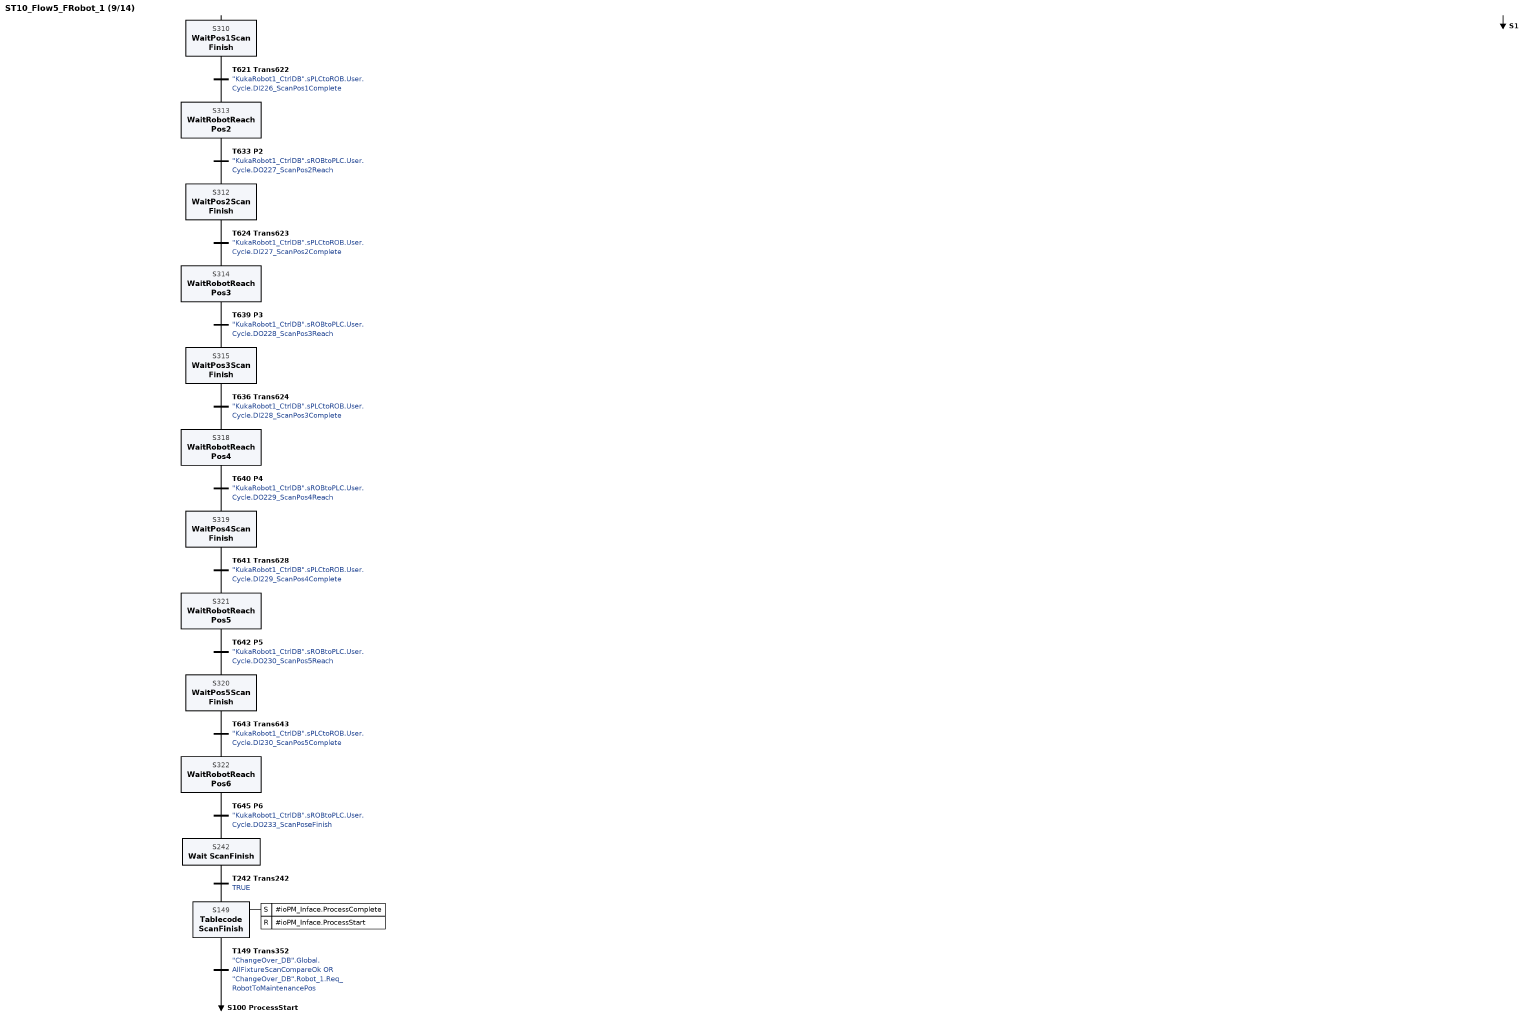
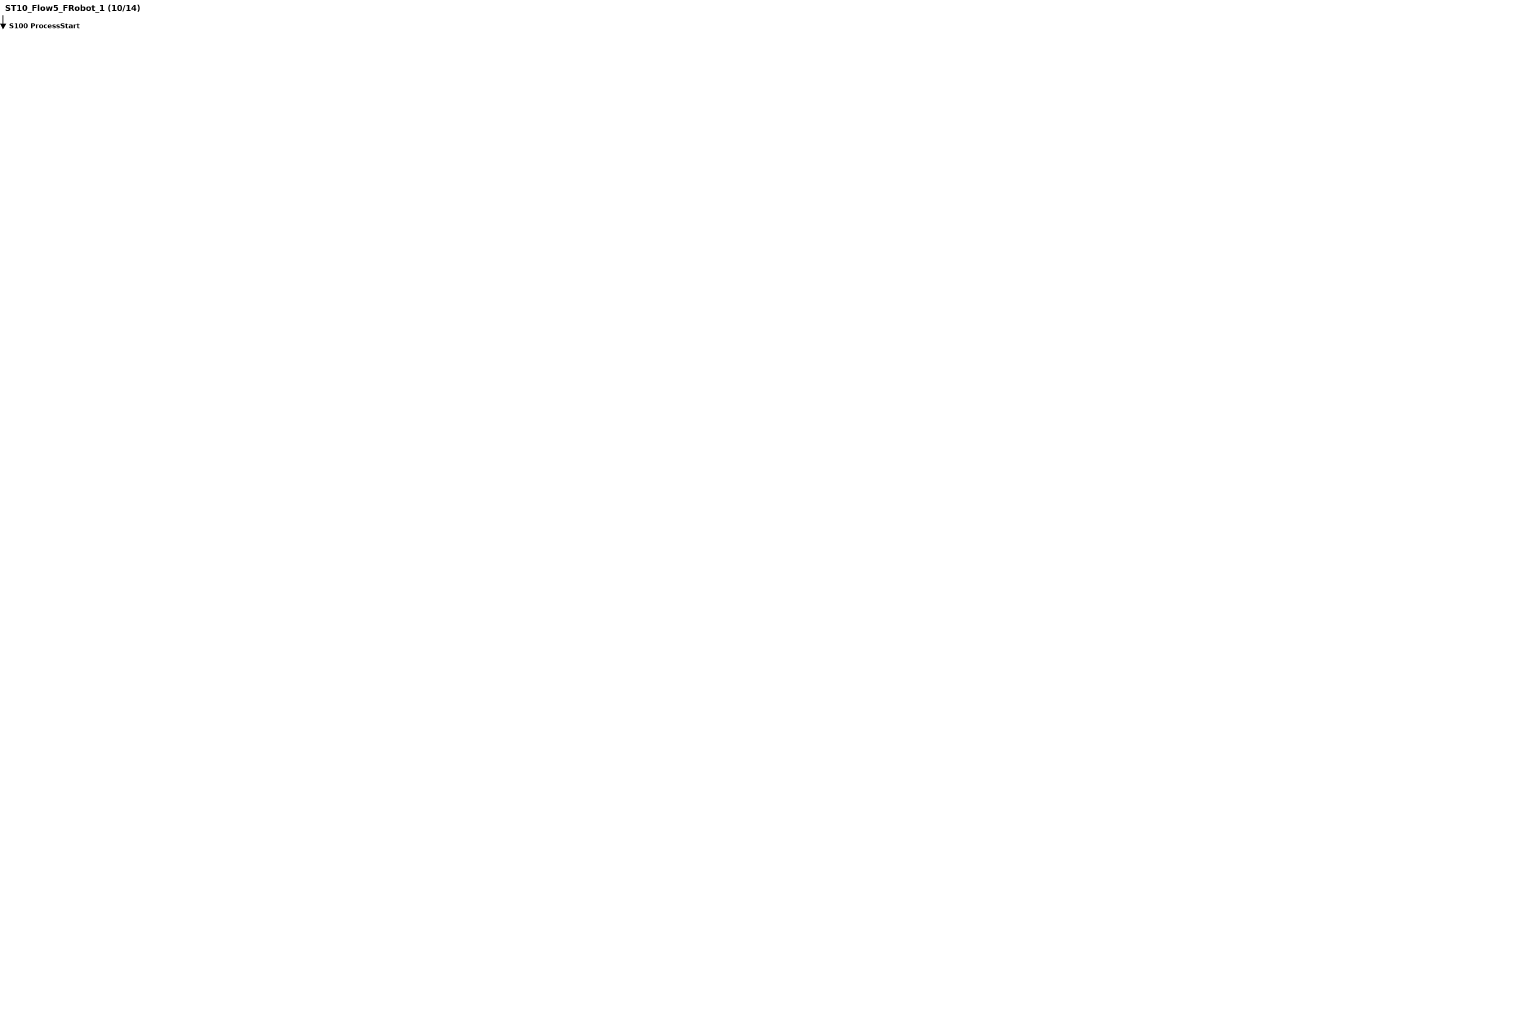
   // permanent pre-instructions
   NETWORK 1
      #TON[10].TON(IN := "AlwaysTRUE" AND "Station_Sys".Alarm.ImmediatelyStop, PT := T#300ms);
      #ioPM_Inface.AlarmImdilyStop := #TON[10].Q;
      #ioPM_Inface.AlarmCycleStop := "AlwaysTRUE" AND "Station_Sys".Alarm.CycleStop;
   NETWORK 2
      IF NOT False THEN
          #sCtrlMode(iSysInface := #iSysInface, ioPM_Inface := #ioPM_Inface, ioGraphCtrl := #RT_DATA.MOP);   // "SysFlowCtrlGraph"
      END_IF;
   NETWORK 3
      #TON[0].TON(IN := "AlwaysTRUE" AND "iA-Rotating product Check", PT := t#500ms);   // 工位11有托盘
      #TON[1].TOF(IN := "AlwaysTRUE" AND NOT "iA-Rotating product Check", PT := T#300ms);   // 工位无托盘
      #TON[2].TON(IN := "AlwaysTRUE", PT := T#300ms);
      #TON[3].TON(IN := "AlwaysTRUE", PT := T#300ms);
      #TON[4].TON(IN := "AlwaysTRUE", PT := T#300ms);
      #TON[5].TON(IN := "AlwaysTRUE", PT := T#300ms);
   NETWORK 4
      #前站站号 := 345;
      #本站站号 := 350;

   // sequencer 1: S01-S99 初始化
   INITIAL_STEP F5_Initial:   // S1, max time T#10S, warning time T#7S
              S    #ioPM_Inface.InitialRun
              R    #ioPM_Inface.InitialOK
              R    #ioPM_Inface.WaitRunning
              R    #ioPM_Inface.Running
              R    #ioPM_Inface.UnPause
              R    "Station_Sys".Cmd.Calibration
              R    "Station_Sys".Cmd.ChangeOver
                   //"ST350_Sys".Cmd.DryRun
              R    "Station_Sys".Cmd.Reserve
              R    "Station_Sys".Cmd.OneCycle
              R    "AutoProcessControl".Robot_1.GluePutFlag
              R    "AutoProcessControl".Robot_1.NGPutFlag
              R    #ioPM_Inface.ProcessComplete
              R    #ioPM_Inface.ProcessStart
          S1  R    "ChangeOver_DB".Robot_1.MaintenancePosReqSelFlag
                   //"Robot_DB".Robot_1.MasteringTest_Req
                   //"Robot_DB".Robot_1.BrakeTest_Req
   END_STEP
   TRANSITION Trans1 FROM F5_Initial TO S2   // T1
      := #iSysInface.Ready;
   END_TRANSITION
   STEP S2:   // S2, max time T#10S, warning time T#7S
   END_STEP
   TRANSITION Trans2 FROM S2 TO S3   // T2
      := TRUE;
   END_TRANSITION
   STEP RobotSpeed:   // S4, max time T#10S, warning time T#7S
              N    "KukaRobot1_CtrlDB".iSpeedValue:=20
   END_STEP
   TRANSITION Trans3 FROM RobotSpeed TO S5_MESInitial   // T3
      := "KukaRobot1_CtrlDB".iSpeedValue = 20;
   END_TRANSITION
   STEP S5_MESInitial:   // S5, max time T#10S, warning time T#7S
   END_STEP
   TRANSITION Trans325 FROM S5_MESInitial TO "RobotManuallyMoved?"   // T4
      := TRUE;
   END_TRANSITION
   STEP S10_InitialFinish:   // S10, max time T#10S, warning time T#7S
              S    #ioPM_Inface.InitialOK
   END_STEP
   TRANSITION Trans102 FROM S10_InitialFinish TO ProcessStart   // T10, jump
      := #ioPM_Inface.Running;
   END_TRANSITION
   STEP S3:   // S3, max time T#10S, warning time T#7S
   END_STEP
   TRANSITION Trans613 FROM S3 TO RobotSpeed   // T607
      := TRUE;
   END_TRANSITION
   STEP S8:   // S8, max time T#10S, warning time T#7S
   END_STEP
   TRANSITION Trans10 FROM S8 TO S9   // T8
      := TRUE;
   END_TRANSITION
   STEP S9:   // S9, max time T#10S, warning time T#7S
   END_STEP
   TRANSITION Trans7 FROM S9 TO S10_InitialFinish   // T9
      := TRUE;
   END_TRANSITION
   STEP "RobotReady?":   // S311, max time T#10S, warning time T#7S
   END_STEP
   TRANSITION Trans606 FROM "RobotReady?" TO RobotStart   // T606
      := "KukaRobot1_CtrlDB".sROBtoPLC.Sys.SO.ALARM_STOP AND "KukaRobot1_CtrlDB".sROBtoPLC.Sys.SO.EXT AND NOT "KukaRobot1_CtrlDB".oStartComplete;
   END_TRANSITION
   STEP RobotStart:   // S316, max time T#10S, warning time T#7S
              N    "KukaRobot1_CtrlDB".ioAutoStart
   END_STEP
   TRANSITION Trans608 FROM RobotStart TO WaitRobotStartHome   // T608
      := "KukaRobot1_CtrlDB".oReady AND "KukaRobot1_CtrlDB".oStartComplete;
   END_TRANSITION
   STEP RobotHome:   // S317, max time T#10S, warning time T#7S
              N    "KukaRobot1_CtrlDB".ioSrartHome
   END_STEP
   TRANSITION Trans609 FROM RobotHome TO RobotAutoCycle   // T609
      := "KukaRobot1_CtrlDB".sROBtoPLC.Sys.SO.IN_HOME AND "KukaRobot1_CtrlDB".sHMI.HomeSeqOK AND "KukaRobot1_CtrlDB".sHMI.WaitForAutoCycleStart AND NOT "KukaRobot1_CtrlDB".sHMI.GoHomeFail;
   END_TRANSITION
   STEP RobotAutoCycle:   // S329, max time T#10S, warning time T#7S
              N    "KukaRobot1_CtrlDB".ioStartAutoCycle
   END_STEP
   TRANSITION Trans612 FROM RobotAutoCycle TO GripStatusCheck   // T610
      := NOT "KukaRobot1_CtrlDB".sHMI.HomeSeqOK AND NOT "KukaRobot1_CtrlDB".sHMI.WaitForAutoCycleStart;
   END_TRANSITION
   STEP GripStatusCheck:   // S330, max time T#10S, warning time T#7S
   END_STEP
   TRANSITION Trans614 FROM GripStatusCheck TO S8   // T611
      := (("AutoProcessData".F_Robot1Grip1.PartStatus = 0) AND ("AutoProcessData".F_Robot1Grip2.PartStatus = 0) AND "iF-ROOBT1Gripper1CylinderInHP" AND NOT "iF-ROOBT1Gripper2Detection") OR (("AutoProcessData".F_Robot1Grip1.PartStatus <> 0) AND NOT "iF-ROOBT1Gripper1CylinderInHP" AND NOT "iF-ROOBT1Gripper1CylinderInWP") OR (("AutoProcessData".F_Robot1Grip2.PartStatus <> 0) AND "iF-ROOBT1Gripper2Detection");
   END_TRANSITION
   TRANSITION Trans616 FROM GripStatusCheck TO Gripe1StatusAlarm   // T613
      := (("AutoProcessData".F_Robot1Grip1.PartStatus = 0) AND NOT "iF-ROOBT1Gripper1CylinderInHP" AND NOT "iF-ROOBT1Gripper1CylinderInWP" AND NOT "ST10Cylinder".Cy[13].In.HomePositionSensor) OR (("AutoProcessData".F_Robot1Grip1.PartStatus <> 0) AND ("iF-ROOBT1Gripper1CylinderInWP" OR "ST10Cylinder".Cy[13].In.HomePositionSensor));
   END_TRANSITION
   TRANSITION Trans617 FROM GripStatusCheck TO Gripe2StatusAlarm   // T612
      := (("AutoProcessData".F_Robot1Grip2.PartStatus = 0) AND "iF-ROOBT1Gripper2Detection" AND NOT "ST10Cylinder".Cy[14].In.HomePositionSensor) OR (("AutoProcessData".F_Robot1Grip2.PartStatus <> 0) AND (NOT "iF-ROOBT1Gripper2Detection" OR "ST10Cylinder".Cy[14].In.HomePositionSensor));
   END_TRANSITION
   STEP Gripe1StatusAlarm:   // S331, max time T#10S, warning time T#7S
          S1  S    "ST10_DeviceError".F.Robot_1.Grip1Error
   END_STEP
   TRANSITION Trans615 FROM Gripe1StatusAlarm TO GripStatusCheck   // T614, jump
      := #iSysInface.Reset;
   END_TRANSITION
   STEP Gripe2StatusAlarm:   // S332, max time T#10S, warning time T#7S
          S1  S    "ST10_DeviceError".F.Robot_1.Grip2Error
   END_STEP
   TRANSITION Trans620 FROM Gripe2StatusAlarm TO GripStatusCheck   // T615, jump
      := #iSysInface.Reset;
   END_TRANSITION
   STEP WaitRobotStartHome:   // S381, max time T#10S, warning time T#7S
   END_STEP
   TRANSITION Trans695 FROM WaitRobotStartHome TO RobotHome   // T695
      := "KukaRobot1_CtrlDB".sROBtoPLC.User.Home.DO161_WaitForHomeSeqStart;
   END_TRANSITION
   STEP "RobotManuallyMoved?":   // S382, max time T#10S, warning time T#7S
   END_STEP
   TRANSITION Trans696 FROM "RobotManuallyMoved?" TO "RobotReady?"   // T696
      := NOT "KukaRobot1_CtrlDB".sPLCtoROB.User.Home.DI169_RobotMoved AND NOT "ST10_DeviceError".F.Robot_1.ManualMoved;
   END_TRANSITION

   // sequencer 2: S100-S199 等待到位
   STEP ProcessStart:   // S100, max time T#10S, warning time T#7S
      // 自动等待开始运行
              R    #ioPM_Inface.InitialRun
              R    #ioPM_Inface.ProcessComplete
              R    #ioPM_Inface.ProcessStart
              S    #ioPM_Inface.InitialOK
              S    #ioPM_Inface.WaitRunning
          S1  N    #ioPM_Inface.ProcessResult:=0
              R    "ST10_GeneralData".FlowControl_Handshake[5].Start
              R    "ST10_GeneralData".FlowControl_Handshake[5].Done
   END_STEP
   TRANSITION Trans200 FROM ProcessStart TO FlagReset   // T100
      := NOT #ioPM_Inface.AlarmCycleStop AND #ioPM_Inface.Running AND NOT #iSysInface.Auto.RunningOver AND (NOT #iSysInface.Auto.OneCycleMode OR (#iSysInface.Auto.OneCycleMode AND #ioPM_Inface.TriggerOneCycle));
   END_TRANSITION
   STEP ScanFixtureCode:   // S110, max time T#10S, warning time T#7S
              R    #ioPM_Inface.ProcessComplete
              S    #ioPM_Inface.ProcessStart
   END_STEP
   TRANSITION Trans625 FROM ScanFixtureCode TO "Tablecode Scan"   // T110, jump
      := TRUE;
   END_TRANSITION
   STEP RobotTaskSelect:   // S333, max time T#10S, warning time T#7S
   END_STEP
   TRANSITION Trans621 FROM RobotTaskSelect TO ScanFixtureCode   // T333
      := NOT "AutoProcessData".GlobalData.Robot1GripperCodeOKFlag AND ("AutoProcessData".F_Robot1Grip1.PartStatus = 0) AND "ST10Cylinder".Cy[13].In.HomePositionSensor AND "AutoProcessControl".Robot_1.GripScanRequest AND NOT "PalletNGData".LoadingNGPallet.OpenFlag AND NOT "ChangeOver_DB".Robot_1.MaintenancePosReqSelFlag AND NOT "Robot_DB".Robot_1.MasteringTest_Req AND NOT "Robot_DB".Robot_1.BrakeTest_Req;
   END_TRANSITION
   TRANSITION Trans630 FROM RobotTaskSelect TO PutBuffer   // T620
      := ("AutoProcessData".F_Robot1Grip1.PartStatus = 100) AND NOT "iF-ROOBT1Gripper1CylinderInHP" AND NOT "iF-ROOBT1Gripper1CylinderInWP" AND NOT "ST10Cylinder".Cy[13].In.HomePositionSensor AND "AutoProcessControl".A_ScanRotary.Robot1PutPrimit AND NOT "PalletNGData".LoadingNGPallet.OpenFlag AND NOT "ChangeOver_DB".Robot_1.MaintenancePosReqSelFlag;
   END_TRANSITION
   TRANSITION Trans632 FROM RobotTaskSelect TO PickTable   // T625
      := (NOT "AutoProcessControl".Robot_1.ClearPart OR (("AutoProcessControl".B_Press_1.Robot1PutRingPrimit OR ("AutoProcessData".A_ScanRotate.PartStatus = 199)) AND "AutoProcessControl".Robot_1.ClearPart)) AND ("AutoProcessData".F_Robot1Grip1.PartStatus = 0) AND "iF-ROOBT1Gripper1CylinderInHP" AND ("AutoProcessData".F_Robot1Grip2.PartStatus = 0) AND NOT "iF-ROOBT1Gripper2Detection" AND "AutoProcessControl".A_Table_1Loading.Robot1PickPrimit AND NOT "PalletNGData".LoadingNGPallet.OpenFlag AND NOT "ChangeOver_DB".Robot_1.MaintenancePosReqSelFlag AND NOT "Robot_DB".Robot_1.MasteringTest_Req AND NOT "Robot_DB".Robot_1.BrakeTest_Req;
   END_TRANSITION
   TRANSITION Trans633 FROM RobotTaskSelect TO ScanRing   // T627
      := ("AutoProcessData".F_Robot1Grip2.PartStatus = 100) AND ("iF-ROOBT1Gripper2Detection" OR "AlwaysTRUE") AND NOT "ST10Cylinder".Cy[14].In.HomePositionSensor AND NOT "KukaRobot1_CtrlDB".sPLCtoROB.User.Cycle.DI261_RingScanReq AND NOT "ChangeOver_DB".Global.ManualModeFlag AND NOT "ChangeOver_DB".Global.ChangeOverSelected AND NOT "PalletNGData".LoadingNGPallet.OpenFlag AND NOT "ChangeOver_DB".Robot_1.MaintenancePosReqSelFlag AND NOT "Robot_DB".Robot_1.MasteringTest_Req AND NOT "Robot_DB".Robot_1.BrakeTest_Req;
   END_TRANSITION
   TRANSITION Trans635 FROM RobotTaskSelect TO PickBuffer   // T629
      := ((("AutoProcessData".F_Robot1Grip2.PartStatus = 199) AND ("iF-ROOBT1Gripper2Detection" OR "AlwaysTRUE")) OR (("AutoProcessData".F_Robot1Grip2.PartStatus = 0) AND ("AutoProcessData".A_ScanRotate.PartStatus = 151))) AND ("AutoProcessData".F_Robot1Grip1.PartStatus = 0) AND "iF-ROOBT1Gripper1CylinderInHP" AND ("AutoProcessData".B_Press1.PartStatus = 0) AND NOT "PalletNGData".LoadingNGPallet.OpenFlag AND "AutoProcessControl".A_ScanRotary.Robot1PickPrimit AND NOT "ChangeOver_DB".Robot_1.MaintenancePosReqSelFlag AND NOT "Robot_DB".Robot_1.MasteringTest_Req AND NOT "Robot_DB".Robot_1.BrakeTest_Req;
   END_TRANSITION
   TRANSITION Trans675 FROM RobotTaskSelect TO "NG1Put_1/Press"   // T674
      := ("AutoProcessData".F_Robot1Grip1.PartStatus >= 250) AND ("AutoProcessData".F_Robot1Grip1.PartStatus <= 260) AND NOT "iF-ROOBT1Gripper1CylinderInHP" AND NOT "iF-ROOBT1Gripper1CylinderInWP" AND NOT "ST10Cylinder".Cy[13].In.HomePositionSensor AND "AutoProcessControl".NG_1.Robot1PutPrimit_1 AND NOT "PalletNGData".LoadingNGPallet.OpenFlag AND NOT "ChangeOver_DB".Robot_1.MaintenancePosReqSelFlag;
   END_TRANSITION
   TRANSITION Trans750 FROM RobotTaskSelect TO "NG1Put_2/ShaftScan"   // T757
      := ("AutoProcessData".F_Robot1Grip1.PartStatus >= 150) AND ("AutoProcessData".F_Robot1Grip1.PartStatus <= 160) AND NOT "iF-ROOBT1Gripper1CylinderInHP" AND NOT "iF-ROOBT1Gripper1CylinderInWP" AND "AutoProcessControl".NG_1.Robot1PutPrimit_2 AND NOT "PalletNGData".LoadingNGPallet.OpenFlag AND NOT "ChangeOver_DB".Robot_1.MaintenancePosReqSelFlag;
   END_TRANSITION
   TRANSITION Trans751 FROM RobotTaskSelect TO "NG1Put_3/RingScan"   // T751
      := ((("AutoProcessData".F_Robot1Grip2.PartStatus >= 150) AND ("AutoProcessData".F_Robot1Grip2.PartStatus <= 160)) OR ("ChangeOver_DB".Global.ManualModeFlag AND ("AutoProcessData".F_Robot1Grip2.PartStatus = 100))) AND ("iF-ROOBT1Gripper2Detection" OR "AlwaysTRUE") AND NOT "ST10Cylinder".Cy[14].In.HomePositionSensor AND "AutoProcessControl".NG_1.Robot1PutPrimit_3 AND NOT "PalletNGData".LoadingNGPallet.OpenFlag AND NOT "ChangeOver_DB".Robot_1.MaintenancePosReqSelFlag;
   END_TRANSITION
   TRANSITION Trans691 FROM RobotTaskSelect TO Grip1SensorError   // T691
      := ((("AutoProcessData".F_Robot1Grip1.PartStatus <> 0) AND "iF-ROOBT1Gripper1CylinderInWP") OR (("AutoProcessData".F_Robot1Grip1.PartStatus = 0) AND NOT "iF-ROOBT1Gripper1CylinderInHP")) AND (#RobotTaskSelect.T > t#3000MS) AND NOT "ChangeOver_DB".Robot_1.MaintenancePosReqSelFlag;
   END_TRANSITION
   TRANSITION Trans692 FROM RobotTaskSelect TO Grip2SensorError   // T692
      := ((("AutoProcessData".F_Robot1Grip2.PartStatus <> 0) AND NOT "iF-ROOBT1Gripper2Detection") OR (("AutoProcessData".F_Robot1Grip2.PartStatus = 0) AND "iF-ROOBT1Gripper2Detection")) AND (#RobotTaskSelect.T > t#3000MS) AND NOT "ChangeOver_DB".Robot_1.MaintenancePosReqSelFlag AND "TON".TON[74].Q;
   END_TRANSITION
   TRANSITION Trans626 FROM RobotTaskSelect TO PickPallet   // T618
      := (NOT "AutoProcessControl".Robot_1.ClearPart OR ("AutoProcessControl".Robot_1.ClearPart AND ("AutoProcessData".F_Robot1Grip2.PartStatus = 199) AND ("AutoProcessData".B_Press1.PartStatus = 0) AND "AutoProcessControl".A_ScanRotary.Robot1PutPrimit) OR "KukaRobot1_CtrlDB".sROBtoPLC.User.Cycle.DO242_SPalletPickFinish) AND NOT "ChangeOver_DB".Global.ChangeOverRequest AND NOT "ChangeOver_DB".Global.ScanFixtureFlag AND "ChangeOver_DB".Global.AllFixtureScanCompareOk AND "AutoProcessData".GlobalData.Robot2GripperCodeOKFlag AND (("AutoProcessData".F_Robot1Grip1.PartStatus = 0) OR ("AutoProcessData".F_Robot1Grip1.PartStatus = 100)) AND "iF-ROOBT1Gripper1CylinderInHP" AND "AutoProcessControl".H_ShafeLine.Robot1PickPrimit AND "AutoProcessControl".A_ScanRotary.Robot1PutPrimit AND NOT "AutoProcessControl".Global.H.EmptyPallet AND ("AutoProcessData".B_Press1.PartStatus <> 199) AND NOT "ChangeOver_DB".Global.ManualModeFlag AND NOT "ChangeOver_DB".Global.ChangeOverSelected AND NOT "PalletNGData".LoadingNGPallet.OpenFlag AND NOT "ChangeOver_DB".Robot_1.MaintenancePosReqSelFlag AND NOT "KukaRobot1_CtrlDB".sROBtoPLC.User.Safety.DO452 AND NOT "KukaRobot1_CtrlDB".sROBtoPLC.User.Safety.DO460 AND (#RobotTaskSelect.T > t#100MS);
   END_TRANSITION
   TRANSITION Trans642 FROM RobotTaskSelect TO PressPick   // T637
      := ("AutoProcessData".F_Robot1Grip1.PartStatus = 0) AND "iF-ROOBT1Gripper1CylinderInHP" AND "AutoProcessControl".B_Press_1.Robot1PickPrimit AND NOT "PalletNGData".LoadingNGPallet.OpenFlag AND NOT "ChangeOver_DB".Robot_1.MaintenancePosReqSelFlag AND NOT "Robot_DB".Robot_1.MasteringTest_Req AND NOT "Robot_DB".Robot_1.BrakeTest_Req;
   END_TRANSITION
   TRANSITION Trans672 FROM RobotTaskSelect TO GluePut   // T672
      := ("AutoProcessData".F_Robot1Grip1.PartStatus = 299) AND NOT "iF-ROOBT1Gripper1CylinderInHP" AND NOT "iF-ROOBT1Gripper1CylinderInWP" AND NOT "ST10Cylinder".Cy[13].In.HomePositionSensor AND "KukaRobot2_CtrlDB".sROBtoPLC.User.Home.DO182_Robot1Area AND NOT "KukaRobot2_CtrlDB".sROBtoPLC.User.Cycle.DO241_PickPalletInside AND NOT "KukaRobot2_CtrlDB".sROBtoPLC.User.Cycle.DO261_ScanPartInside AND NOT "KukaRobot2_CtrlDB".sROBtoPLC.User.Cycle.DO265_GluePutInside AND NOT "KukaRobot2_CtrlDB".sROBtoPLC.User.Cycle.DO269_GluePickInside AND NOT "AutoProcessControl".Robot_2.PalletPickFlag AND NOT "AutoProcessControl".Robot_2.MagnetScanFlag AND NOT "AutoProcessControl".Robot_2.GluePutFlag AND NOT "AutoProcessControl".Robot_2.GluePickFlag AND "AutoProcessControl".C_Glue.Robot1PutPrimit AND NOT "PalletNGData".LoadingNGPallet.OpenFlag AND NOT "ChangeOver_DB".Robot_1.MaintenancePosReqSelFlag AND NOT "Robot_DB".Robot_1.MasteringTest_Req AND NOT "Robot_DB".Robot_1.BrakeTest_Req;
   END_TRANSITION
   TRANSITION Trans637 FROM RobotTaskSelect TO PressShaftPut   // T631
      := ("AutoProcessData".F_Robot1Grip1.PartStatus = 199) AND NOT "iF-ROOBT1Gripper1CylinderInHP" AND NOT "iF-ROOBT1Gripper1CylinderInWP" AND NOT "ST10Cylinder".Cy[13].In.HomePositionSensor AND ("AutoProcessData".F_Robot1Grip2.PartStatus = 199) AND ("iF-ROOBT1Gripper2Detection" OR "AlwaysTRUE") AND NOT "ST10Cylinder".Cy[14].In.HomePositionSensor AND "AutoProcessControl".B_Press_1.Robot1PutShaftPrimit AND NOT "PalletNGData".LoadingNGPallet.OpenFlag AND NOT "ChangeOver_DB".Robot_1.MaintenancePosReqSelFlag AND NOT "Robot_DB".Robot_1.MasteringTest_Req AND NOT "Robot_DB".Robot_1.BrakeTest_Req;
   END_TRANSITION
   TRANSITION Trans640 FROM RobotTaskSelect TO PressRingPut   // T634
      := ("AutoProcessData".F_Robot1Grip2.PartStatus = 199) AND ("iF-ROOBT1Gripper2Detection" OR "AlwaysTRUE") AND NOT "ST10Cylinder".Cy[14].In.HomePositionSensor AND ("AutoProcessData".F_Robot1Grip1.PartStatus = 0) AND "iF-ROOBT1Gripper1CylinderInHP" AND "ST10Cylinder".Cy[13].In.HomePositionSensor AND "AutoProcessControl".B_Press_1.Robot1PutRingPrimit AND NOT "PalletNGData".LoadingNGPallet.OpenFlag AND NOT "ChangeOver_DB".Robot_1.MaintenancePosReqSelFlag AND NOT "Robot_DB".Robot_1.MasteringTest_Req AND NOT "Robot_DB".Robot_1.BrakeTest_Req;
   END_TRANSITION
   TRANSITION Trans711 FROM RobotTaskSelect TO Maintenance   // T638
      := (("iF-ROOBT1Gripper1CylinderInHP" AND NOT "iF-ROOBT1Gripper2Detection" AND ("AutoProcessData".F_Robot1Grip2.PartStatus = 0) AND ("AutoProcessData".F_Robot1Grip1.PartStatus = 0) AND "ChangeOver_DB".Robot_1.Req_RobotToMaintenancePos AND NOT "PalletNGData".LoadingNGPallet.OpenFlag) OR (NOT "AutoProcessControl".Robot_1.MaintenanceRequest AND "ChangeOver_DB".Robot_1.HMI_MaintenancePosActive)) AND NOT "Robot_DB".Robot_1.MasteringTest_Req AND NOT "Robot_DB".Robot_1.BrakeTest_Req;
   END_TRANSITION
   TRANSITION Trans900 FROM RobotTaskSelect TO Masref_test   // T900
      := ("AutoProcessData".F_Robot1Grip1.PartStatus = 0) AND "iF-ROOBT1Gripper1CylinderInHP" AND "Robot_DB".Robot_1.MasteringTest_Req;
   END_TRANSITION
   TRANSITION Trans901 FROM RobotTaskSelect TO Brake_Test   // T901
      := ("AutoProcessData".F_Robot1Grip1.PartStatus = 0) AND "iF-ROOBT1Gripper1CylinderInHP" AND "Robot_DB".Robot_1.BrakeTest_Req;
   END_TRANSITION
   STEP PressPick:   // S150, max time T#10S, warning time T#7S
              R    #ioPM_Inface.ProcessComplete
              S    #ioPM_Inface.ProcessStart
   END_STEP
   TRANSITION Trans641 FROM PressPick TO PressPickProcess   // T150, jump
      := TRUE;
   END_TRANSITION
   STEP PutBuffer:   // S120, max time T#10S, warning time T#7S
              R    #ioPM_Inface.ProcessComplete
              S    #ioPM_Inface.ProcessStart
   END_STEP
   TRANSITION Trans629 FROM PutBuffer TO PutBufferProcess   // T120, jump
      := TRUE;
   END_TRANSITION
   STEP PickTable:   // S130, max time T#10S, warning time T#7S
              R    #ioPM_Inface.ProcessComplete
              S    #ioPM_Inface.ProcessStart
   END_STEP
   TRANSITION Trans631 FROM PickTable TO PickTableProcess   // T130, jump
      := TRUE;
   END_TRANSITION
   STEP ScanRing:   // S135, max time T#10S, warning time T#7S
              R    #ioPM_Inface.ProcessComplete
              S    #ioPM_Inface.ProcessStart
   END_STEP
   TRANSITION Trans634 FROM ScanRing TO ScanRingProcess   // T135, jump
      := TRUE;
   END_TRANSITION
   STEP PickBuffer:   // S125, max time T#10S, warning time T#7S
              R    #ioPM_Inface.ProcessComplete
              S    #ioPM_Inface.ProcessStart
   END_STEP
   TRANSITION Trans636 FROM PickBuffer TO PickBufferProcess   // T125, jump
      := TRUE;
   END_TRANSITION
   STEP "NG1Put_1/Press":   // S160, max time T#10S, warning time T#7S
              S    "AutoProcessControl".Robot_1.NGPutFlag
              R    #ioPM_Inface.ProcessComplete
              S    #ioPM_Inface.ProcessStart
   END_STEP
   TRANSITION Trans676 FROM "NG1Put_1/Press" TO "NG PutProcess"   // T160, jump
      := "AutoProcessControl".Robot_1.NGPutFlag;
   END_TRANSITION
   STEP "NG1Put_2/ShaftScan":   // S165, max time T#10S, warning time T#7S
              S    "AutoProcessControl".Robot_1.NGPutFlag
              R    #ioPM_Inface.ProcessComplete
              S    #ioPM_Inface.ProcessStart
   END_STEP
   TRANSITION Trans677 FROM "NG1Put_2/ShaftScan" TO "NG 2 PutProcess"   // T165, jump
      := "AutoProcessControl".Robot_1.NGPutFlag;
   END_TRANSITION
   STEP "NG1Put_3/RingScan":   // S170, max time T#10S, warning time T#7S
              S    "AutoProcessControl".Robot_1.NGPutFlag
              R    #ioPM_Inface.ProcessComplete
              S    #ioPM_Inface.ProcessStart
   END_STEP
   TRANSITION Trans679 FROM "NG1Put_3/RingScan" TO "NG 3 PutProcess"   // T170, jump
      := "AutoProcessControl".Robot_1.NGPutFlag;
   END_TRANSITION
   STEP Grip1SensorError:   // S379, max time T#10S, warning time T#7S
   END_STEP
   TRANSITION Trans693 FROM Grip1SensorError TO RobotTaskSelect   // T693, jump
      := #iSysInface.Reset;
   END_TRANSITION
   STEP Grip2SensorError:   // S380, max time T#10S, warning time T#7S
   END_STEP
   TRANSITION Trans694 FROM Grip2SensorError TO RobotTaskSelect   // T694, jump
      := #iSysInface.Reset;
   END_TRANSITION
   STEP PressRingPut:   // S145, max time T#10S, warning time T#7S
              R    #ioPM_Inface.ProcessComplete
              S    #ioPM_Inface.ProcessStart
   END_STEP
   TRANSITION Trans639 FROM PressRingPut TO PressRingPutProcess   // T145, jump
      := TRUE;
   END_TRANSITION
   STEP PickPallet:   // S115, max time T#10S, warning time T#7S
              R    #ioPM_Inface.ProcessComplete
              S    #ioPM_Inface.ProcessStart
   END_STEP
   TRANSITION Trans627 FROM PickPallet TO PickPalletProcess   // T115, jump
      := TRUE;
   END_TRANSITION
   STEP GluePut:   // S155, max time T#10S, warning time T#7S
              S    "AutoProcessControl".Robot_1.GluePutFlag
              R    #ioPM_Inface.ProcessComplete
              S    #ioPM_Inface.ProcessStart
   END_STEP
   TRANSITION Trans649 FROM GluePut TO GluePutProcess   // T155, jump
      := "AutoProcessControl".Robot_1.GluePutFlag;
   END_TRANSITION
   STEP PressShaftPut:   // S140, max time T#10S, warning time T#7S
              R    #ioPM_Inface.ProcessComplete
              S    #ioPM_Inface.ProcessStart
   END_STEP
   TRANSITION Trans638 FROM PressShaftPut TO PressShaftPutProcess   // T140, jump
      := TRUE;
   END_TRANSITION
   STEP FlagReset:   // S383, max time T#10S, warning time T#7S
              R    "AutoProcessControl".Robot_1.GluePutFlag
              R    "AutoProcessControl".Robot_1.NGPutFlag
   END_STEP
   TRANSITION Trans697 FROM FlagReset TO RobotTaskSelect   // T697
      := NOT "AutoProcessControl".Robot_1.GluePutFlag AND NOT "AutoProcessControl".Robot_1.NGPutFlag;
   END_TRANSITION
   STEP Maintenance:   // S131, max time T#10S, warning time T#7S
              R    #ioPM_Inface.ProcessComplete
              S    #ioPM_Inface.ProcessStart
   END_STEP
   TRANSITION Trans710 FROM Maintenance TO "Maintenance Pos"   // T131, jump
      := TRUE;
   END_TRANSITION
   STEP Masref_test:   // S132, max time T#10S, warning time T#7S
              R    #ioPM_Inface.ProcessComplete
              S    #ioPM_Inface.ProcessStart
   END_STEP
   TRANSITION Trans712 FROM Masref_test TO MasteringTest_Req   // T132, jump
      := TRUE;
   END_TRANSITION
   STEP Brake_Test:   // S133, max time T#10S, warning time T#7S
              R    #ioPM_Inface.ProcessComplete
              S    #ioPM_Inface.ProcessStart
   END_STEP
   TRANSITION Trans713 FROM Brake_Test TO BrakeTest_Req   // T133, jump
      := TRUE;
   END_TRANSITION

   // sequencer 3
   STEP "Tablecode Scan":   // S200, max time T#10S, warning time T#7S
   END_STEP
   TRANSITION Trans147 FROM "Tablecode Scan" TO StartRobotScanGripperCode   // T200
      := NOT "KukaRobot2_CtrlDB".sROBtoPLC.User.Cycle.DO305_GripScanInside AND "KukaRobot2_CtrlDB".sROBtoPLC.Sys.SO.I_O_ACTCONF AND "AutoProcessControl".Robot_1.GripScanRequest;
   END_TRANSITION
   STEP WaitPos4ScanFinish:   // S319, max time T#10S, warning time T#7S
   END_STEP
   TRANSITION Trans628 FROM WaitPos4ScanFinish TO WaitRobotReachPos5   // T641
      := "KukaRobot1_CtrlDB".sPLCtoROB.User.Cycle.DI229_ScanPos4Complete;
   END_TRANSITION
   STEP WaitRobotReachPos3:   // S314, max time T#10S, warning time T#7S
   END_STEP
   TRANSITION P3 FROM WaitRobotReachPos3 TO WaitPos3ScanFinish   // T639
      := "KukaRobot1_CtrlDB".sROBtoPLC.User.Cycle.DO228_ScanPos3Reach;
   END_TRANSITION
   STEP WaitRobotReachPos5:   // S321, max time T#10S, warning time T#7S
   END_STEP
   TRANSITION P5 FROM WaitRobotReachPos5 TO WaitPos5ScanFinish   // T642
      := "KukaRobot1_CtrlDB".sROBtoPLC.User.Cycle.DO230_ScanPos5Reach;
   END_TRANSITION
   STEP WaitPos5ScanFinish:   // S320, max time T#10S, warning time T#7S
   END_STEP
   TRANSITION Trans643 FROM WaitPos5ScanFinish TO WaitRobotReachPos6   // T643
      := "KukaRobot1_CtrlDB".sPLCtoROB.User.Cycle.DI230_ScanPos5Complete;
   END_TRANSITION
   STEP WaitPos3ScanFinish:   // S315, max time T#10S, warning time T#7S
   END_STEP
   TRANSITION Trans624 FROM WaitPos3ScanFinish TO WaitRobotReachPos4   // T636
      := "KukaRobot1_CtrlDB".sPLCtoROB.User.Cycle.DI228_ScanPos3Complete;
   END_TRANSITION
   STEP WaitRobotReachPos2:   // S313, max time T#10S, warning time T#7S
   END_STEP
   TRANSITION P2 FROM WaitRobotReachPos2 TO WaitPos2ScanFinish   // T633
      := "KukaRobot1_CtrlDB".sROBtoPLC.User.Cycle.DO227_ScanPos2Reach;
   END_TRANSITION
   STEP StartRobotScanFixtureCode:   // S308, max time T#10S, warning time T#7S
              N    "KukaRobot1_CtrlDB".sPLCtoROB.User.Cycle.DI225_ScanPosReq
   END_STEP
   TRANSITION Trans605 FROM StartRobotScanFixtureCode TO WaitRobotReachPos1   // T605
      := "KukaRobot1_CtrlDB".sROBtoPLC.User.Cycle.DO225_ScanPosInside AND NOT "KukaRobot1_CtrlDB".sROBtoPLC.User.Cycle.DO233_ScanPoseFinish;
   END_TRANSITION
   STEP WaitRobotReachPos4:   // S318, max time T#10S, warning time T#7S
   END_STEP
   TRANSITION P4 FROM WaitRobotReachPos4 TO WaitPos4ScanFinish   // T640
      := "KukaRobot1_CtrlDB".sROBtoPLC.User.Cycle.DO229_ScanPos4Reach;
   END_TRANSITION
   STEP WaitPos1ScanFinish:   // S310, max time T#10S, warning time T#7S
   END_STEP
   TRANSITION Trans622 FROM WaitPos1ScanFinish TO WaitRobotReachPos2   // T621
      := "KukaRobot1_CtrlDB".sPLCtoROB.User.Cycle.DI226_ScanPos1Complete;
   END_TRANSITION
   STEP WaitRobotReachPos1:   // S309, max time T#10S, warning time T#7S
   END_STEP
   TRANSITION P1 FROM WaitRobotReachPos1 TO WaitPos1ScanFinish   // T617
      := "KukaRobot1_CtrlDB".sROBtoPLC.User.Cycle.DO226_ScanPos1Reach;
   END_TRANSITION
   STEP WaitPos2ScanFinish:   // S312, max time T#10S, warning time T#7S
   END_STEP
   TRANSITION Trans623 FROM WaitPos2ScanFinish TO WaitRobotReachPos3   // T624
      := "KukaRobot1_CtrlDB".sPLCtoROB.User.Cycle.DI227_ScanPos2Complete;
   END_TRANSITION
   STEP WaitRobotReachPos6:   // S322, max time T#10S, warning time T#7S
   END_STEP
   TRANSITION P6 FROM WaitRobotReachPos6 TO "Wait ScanFinish"   // T645
      := "KukaRobot1_CtrlDB".sROBtoPLC.User.Cycle.DO233_ScanPoseFinish;
   END_TRANSITION
   STEP "Wait ScanFinish":   // S242, max time T#10S, warning time T#7S
   END_STEP
   TRANSITION Trans242 FROM "Wait ScanFinish" TO "Tablecode ScanFinish"   // T242
      := TRUE;
   END_TRANSITION
   STEP "Tablecode ScanFinish":   // S149, max time T#10S, warning time T#7S
              S    #ioPM_Inface.ProcessComplete
              R    #ioPM_Inface.ProcessStart
   END_STEP
   TRANSITION Trans352 FROM "Tablecode ScanFinish" TO ProcessStart   // T149, jump
      := "ChangeOver_DB".Global.AllFixtureScanCompareOk OR "ChangeOver_DB".Robot_1.Req_RobotToMaintenancePos;
   END_TRANSITION
   STEP StartRobotScanGripperCode:   // S334, max time T#10S, warning time T#7S
              N    "KukaRobot1_CtrlDB".sPLCtoROB.User.Cycle.DI305_GripScan
   END_STEP
   TRANSITION Trans684 FROM StartRobotScanGripperCode TO RobotScanGripperReachPos1   // T616
      := "KukaRobot1_CtrlDB".sROBtoPLC.User.Cycle.DO305_GripScanInside AND NOT "KukaRobot1_CtrlDB".sROBtoPLC.User.Cycle.DO306_GripScanFinish;
   END_TRANSITION
   STEP RobotScanGripperReachPos1:   // S335, max time T#10S, warning time T#7S
   END_STEP
   TRANSITION Trans685 FROM RobotScanGripperReachPos1 TO WaitGripperPos1ScanFinish   // T619
      := "KukaRobot1_CtrlDB".sROBtoPLC.User.Cycle.DO307_ScanPos1Reach;
   END_TRANSITION
   STEP WaitGripperPos1ScanFinish:   // S336, max time T#10S, warning time T#7S
   END_STEP
   TRANSITION Trans686 FROM WaitGripperPos1ScanFinish TO RobotScanGripperReachPos2   // T622
      := "KukaRobot1_CtrlDB".sPLCtoROB.User.Cycle.DI306_ScanPartComplete;
   END_TRANSITION
   STEP RobotScanGripperReachPos2:   // S337, max time T#10S, warning time T#7S
   END_STEP
   TRANSITION Trans687 FROM RobotScanGripperReachPos2 TO WaitGripperPos2ScanFinish   // T623
      := "KukaRobot1_CtrlDB".sROBtoPLC.User.Cycle.DO308_ScanPos2Reach;
   END_TRANSITION
   STEP WaitGripperPos2ScanFinish:   // S338, max time T#10S, warning time T#7S
   END_STEP
   TRANSITION Trans688 FROM WaitGripperPos2ScanFinish TO RobotScanGripperReachPos3   // T626
      := "KukaRobot1_CtrlDB".sPLCtoROB.User.Cycle.DI306_ScanPartComplete;
   END_TRANSITION
   STEP RobotScanGripperReachPos3:   // S339, max time T#10S, warning time T#7S
   END_STEP
   TRANSITION Trans689 FROM RobotScanGripperReachPos3 TO WaitGripperPos3ScanFinish   // T628
      := "KukaRobot1_CtrlDB".sROBtoPLC.User.Cycle.DO309_ScanPos3Reach;
   END_TRANSITION
   STEP WaitGripperPos3ScanFinish:   // S340, max time T#10S, warning time T#7S
   END_STEP
   TRANSITION Trans690 FROM WaitGripperPos3ScanFinish TO RobotScanGripperReachPos4   // T630
      := "KukaRobot1_CtrlDB".sPLCtoROB.User.Cycle.DI306_ScanPartComplete;
   END_TRANSITION
   STEP RobotScanGripperReachPos4:   // S341, max time T#10S, warning time T#7S
   END_STEP
   TRANSITION Trans698 FROM RobotScanGripperReachPos4 TO WaitGripperPos4ScanFinish   // T632
      := "KukaRobot1_CtrlDB".sROBtoPLC.User.Cycle.DO310_ScanPos4Reach;
   END_TRANSITION
   STEP WaitGripperPos4ScanFinish:   // S342, max time T#10S, warning time T#7S
   END_STEP
   TRANSITION Trans699 FROM WaitGripperPos4ScanFinish TO StartRobotScanFixtureCode   // T635
      := "KukaRobot1_CtrlDB".sROBtoPLC.User.Cycle.DO306_GripScanFinish AND "AutoProcessControl".Fixture1Code.Robot1CodeReadReq;
   END_TRANSITION

   // sequencer 4
   STEP PickPalletProcess:   // S250, max time T#10S, warning time T#7S
   END_STEP
   TRANSITION Trans150 FROM PickPalletProcess TO DataClear   // T250
      := TRUE;
   END_TRANSITION
   STEP StartRobotPickPalletShaft:   // S326, max time T#10S, warning time T#7S
              N    "KukaRobot1_CtrlDB".sPLCtoROB.User.Cycle.DI241_PickShaftPalletReq
   END_STEP
   TRANSITION Trans607 FROM StartRobotPickPalletShaft TO WaitRobotGripHaveStatus   // T648
      := "KukaRobot1_CtrlDB".sROBtoPLC.User.Cycle.DO241_SPalletPickInside AND NOT "KukaRobot1_CtrlDB".sROBtoPLC.User.Cycle.DO242_SPalletPickFinish;
   END_TRANSITION
   STEP WaitRobotFinish:   // S327, max time T#10S, warning time T#7S
   END_STEP
   TRANSITION P8 FROM WaitRobotFinish TO PickPalletFinish   // T327
      := "KukaRobot1_CtrlDB".sROBtoPLC.User.Cycle.DO242_SPalletPickFinish;
   END_TRANSITION
   STEP PickPalletFinish:   // S299, max time T#10S, warning time T#7S
              S    #ioPM_Inface.ProcessComplete
              R    #ioPM_Inface.ProcessStart
   END_STEP
   TRANSITION Trans654 FROM PickPalletFinish TO ProcessStart   // T299, jump
      := TRUE;
   END_TRANSITION
   STEP WaitRobotGripHaveStatus:   // S346, max time T#10S, warning time T#7S
   END_STEP
   TRANSITION Trans655 FROM WaitRobotGripHaveStatus TO Grip1PartStatus   // T655
      := ("KukaRobot1_CtrlDB".sROBtoPLC.User.Public.GO5_RobGrip1Status <> 0) OR "KukaRobot1_CtrlDB".sROBtoPLC.User.Cycle.DO242_SPalletPickFinish;
   END_TRANSITION
   STEP Grip1PartStatus:   // S243, max time T#10S, warning time T#7S
      interlock C := NOT "iF-ROOBT1Gripper1CylinderInHP" AND NOT "iF-ROOBT1Gripper1CylinderInWP";
      (C)     N    "AutoProcessData".F_Robot1Grip1.PartStatus:=100
   END_STEP
   TRANSITION Trans243 FROM Grip1PartStatus TO WaitRobotFinish   // T243
      := (NOT "iF-ROOBT1Gripper1CylinderInHP" AND NOT "iF-ROOBT1Gripper1CylinderInWP" AND ("AutoProcessData".F_Robot1Grip1.PartStatus = 100)) OR ("iF-ROOBT1Gripper1CylinderInHP" AND (#Grip1PartStatus.T > t#500MS));
   END_TRANSITION
   STEP DataClear:   // S252, max time T#10S, warning time T#7S
      // CJ - check
          S1  N    "AutoProcessData".F_Robot1Grip1:="AutoProcessData".ClearData
   END_STEP
   TRANSITION Trans253 FROM DataClear TO StartRobotPickPalletShaft   // T253
      := TRUE;
   END_TRANSITION

   // sequencer 5
   STEP PutBufferProcess:   // S300, max time T#10S, warning time T#7S
   END_STEP
   TRANSITION Trans300 FROM PutBufferProcess TO StartRobotPutBuffer   // T300
      := TRUE;
   END_TRANSITION
   STEP DataMove:   // S253, max time T#10S, warning time T#7S
          S1  N    "AutoProcessData".A_ScanRotate:="AutoProcessData".F_Robot1Grip1
          S1  N    "AutoProcessData".F_Robot1Grip1:="AutoProcessData".ClearData
   END_STEP
   TRANSITION Trans254 FROM DataMove TO WaitRobotFinish_1   // T254
      := #DataMove.T > t#100MS;
   END_TRANSITION
   STEP StartRobotPutBuffer:   // S328, max time T#10S, warning time T#7S
              N    "KukaRobot1_CtrlDB".sPLCtoROB.User.Cycle.DI249_ShaftScanPutReq
   END_STEP
   TRANSITION Trans610 FROM StartRobotPutBuffer TO WaitRobotGripHaveStatus_1   // T328
      := "KukaRobot1_CtrlDB".sROBtoPLC.User.Cycle.DO249_ShaftScanPutInside AND NOT "KukaRobot1_CtrlDB".sROBtoPLC.User.Cycle.DO250_ShaftScanPutFinish;
   END_TRANSITION
   STEP WaitRobotFinish_1:   // S343, max time T#10S, warning time T#7S
   END_STEP
   TRANSITION P9 FROM WaitRobotFinish_1 TO PutBufferFinish_1   // T651
      := "KukaRobot1_CtrlDB".sROBtoPLC.User.Cycle.DO250_ShaftScanPutFinish;
   END_TRANSITION
   STEP PutBufferFinish_1:   // S349, max time T#10S, warning time T#7S
              S    #ioPM_Inface.ProcessComplete
              R    #ioPM_Inface.ProcessStart
   END_STEP
   TRANSITION Trans656 FROM PutBufferFinish_1 TO ProcessStart   // T349, jump
      := TRUE;
   END_TRANSITION
   STEP WaitRobotGripHaveStatus_1:   // S347, max time T#10S, warning time T#7S
   END_STEP
   TRANSITION Trans657 FROM WaitRobotGripHaveStatus_1 TO DataMove   // T656
      := "KukaRobot1_CtrlDB".sROBtoPLC.User.Public.GO5_RobGrip1Status = 0;
   END_TRANSITION

   // sequencer 6
   STEP PickBufferProcess:   // S350, max time T#10S, warning time T#7S
   END_STEP
   TRANSITION Trans350 FROM PickBufferProcess TO StartRobotPickBuffer   // T350
      := TRUE;
   END_TRANSITION
   STEP DataMove_1:   // S255, max time T#10S, warning time T#7S
          S1  N    "AutoProcessData".F_Robot1Grip1:="AutoProcessData".A_ScanRotate
          S1  N    "AutoProcessData".A_ScanRotate:="AutoProcessData".ClearData
   END_STEP
   TRANSITION Trans256 FROM DataMove_1 TO WaitRobotFinish_2   // T256
      := #DataMove_1.T > t#100MS;
   END_TRANSITION
   STEP StartRobotPickBuffer:   // S344, max time T#10S, warning time T#7S
              N    "KukaRobot1_CtrlDB".sPLCtoROB.User.Cycle.DI253_ShaftScanPickReq
   END_STEP
   TRANSITION Trans611 FROM StartRobotPickBuffer TO WaitRobotGripHaveStatus_2   // T652
      := "KukaRobot1_CtrlDB".sROBtoPLC.User.Cycle.DO253_SScanPickInside AND NOT "KukaRobot1_CtrlDB".sROBtoPLC.User.Cycle.DO254_SScanPickFinish;
   END_TRANSITION
   STEP WaitRobotFinish_2:   // S345, max time T#10S, warning time T#7S
   END_STEP
   TRANSITION P10 FROM WaitRobotFinish_2 TO PickBufferFinish   // T653
      := "KukaRobot1_CtrlDB".sROBtoPLC.User.Cycle.DO254_SScanPickFinish;
   END_TRANSITION
   STEP PickBufferFinish:   // S399, max time T#10S, warning time T#7S
              S    #ioPM_Inface.ProcessComplete
              R    #ioPM_Inface.ProcessStart
   END_STEP
   TRANSITION Trans658 FROM PickBufferFinish TO ProcessStart   // T399, jump
      := TRUE;
   END_TRANSITION
   STEP WaitRobotGripHaveStatus_2:   // S348, max time T#10S, warning time T#7S
   END_STEP
   TRANSITION Trans659 FROM WaitRobotGripHaveStatus_2 TO DataMove_1   // T657
      := "KukaRobot1_CtrlDB".sROBtoPLC.User.Public.GO5_RobGrip1Status <> 0;
   END_TRANSITION

   // sequencer 7
   STEP PickTableProcess:   // S400, max time T#10S, warning time T#7S
   END_STEP
   TRANSITION Trans400 FROM PickTableProcess TO "Data Clear_2"   // T400
      := TRUE;
   END_TRANSITION
   STEP Grip2PartStatus:   // S244, max time T#10S, warning time T#7S
              N    "AutoProcessData".F_Robot1Grip2.PartStatus:=100
   END_STEP
   TRANSITION Trans244 FROM Grip2PartStatus TO WaitRobotFinish_3   // T244
      := "AutoProcessData".F_Robot1Grip2.PartStatus = 100;
   END_TRANSITION
   STEP StartRobotPickTable:   // S352, max time T#10S, warning time T#7S
              N    "KukaRobot1_CtrlDB".sPLCtoROB.User.Cycle.DI257_TableRingPickReq
   END_STEP
   TRANSITION Trans618 FROM StartRobotPickTable TO WaitRobotGripHaveStatus_3   // T654
      := "KukaRobot1_CtrlDB".sROBtoPLC.User.Cycle.DO257_TablePickInside AND NOT "KukaRobot1_CtrlDB".sROBtoPLC.User.Cycle.DO258_TablePickFinish;
   END_TRANSITION
   STEP WaitRobotFinish_3:   // S353, max time T#10S, warning time T#7S
   END_STEP
   TRANSITION P11 FROM WaitRobotFinish_3 TO PickTableProcessFinish   // T658
      := "KukaRobot1_CtrlDB".sROBtoPLC.User.Cycle.DO258_TablePickFinish;
   END_TRANSITION
   STEP PickTableProcessFinish:   // S449, max time T#10S, warning time T#7S
              S    #ioPM_Inface.ProcessComplete
              R    #ioPM_Inface.ProcessStart
   END_STEP
   TRANSITION Trans660 FROM PickTableProcessFinish TO ProcessStart   // T449, jump
      := TRUE;
   END_TRANSITION
   STEP WaitRobotGripHaveStatus_3:   // S354, max time T#10S, warning time T#7S
   END_STEP
   TRANSITION Trans661 FROM WaitRobotGripHaveStatus_3 TO Grip2PartStatus   // T659
      := "KukaRobot1_CtrlDB".sROBtoPLC.User.Public.GO6_RobGrip2Status <> 0;
   END_TRANSITION
   STEP "Data Clear_2":   // S258, max time T#10S, warning time T#7S
          S1  N    "AutoProcessData".F_Robot1Grip2:="AutoProcessData".ClearData
   END_STEP
   TRANSITION Trans259 FROM "Data Clear_2" TO StartRobotPickTable   // T259
      := #"Data Clear_2".T > t#100MS;
   END_TRANSITION

   // sequencer 8
   STEP ScanRingProcess:   // S450, max time T#10S, warning time T#7S
   END_STEP
   TRANSITION Trans450 FROM ScanRingProcess TO StartRobotScanRing   // T450
      := TRUE;
   END_TRANSITION
   STEP CheckScanReady:   // S245, max time T#10S, warning time T#7S
   END_STEP
   TRANSITION Trans245 FROM CheckScanReady TO ScanStart   // T245
      := "KeyenceSR1000Ctrl_804A1DB".oReady;
   END_TRANSITION
   STEP StartRobotScanRing:   // S355, max time T#10S, warning time T#7S
              N    "KukaRobot1_CtrlDB".sPLCtoROB.User.Cycle.DI261_RingScanReq
   END_STEP
   TRANSITION Trans619 FROM StartRobotScanRing TO WaitRobotReachScanPos   // T660
      := "KukaRobot1_CtrlDB".sROBtoPLC.User.Cycle.DO261_RingScanInside AND NOT "KukaRobot1_CtrlDB".sROBtoPLC.User.Cycle.DO262_RingScanFinish;
   END_TRANSITION
   STEP WaitRobotFinish_4:   // S356, max time T#10S, warning time T#7S
              N    "KukaRobot1_CtrlDB".sPLCtoROB.User.Cycle.DI262_RingScanComplete
   END_STEP
   TRANSITION P12 FROM WaitRobotFinish_4 TO ScanRingProcessFinish   // T661
      := "KukaRobot1_CtrlDB".sROBtoPLC.User.Cycle.DO262_RingScanFinish;
   END_TRANSITION
   STEP ScanRingProcessFinish:   // S499, max time T#10S, warning time T#7S
              S    #ioPM_Inface.ProcessComplete
              R    #ioPM_Inface.ProcessStart
   END_STEP
   TRANSITION Trans662 FROM ScanRingProcessFinish TO ProcessStart   // T499, jump
      := TRUE;
   END_TRANSITION
   STEP WaitRobotReachScanPos:   // S357, max time T#10S, warning time T#7S
   END_STEP
   TRANSITION Trans663 FROM WaitRobotReachScanPos TO CheckScanReady   // T662
      := "KukaRobot1_CtrlDB".sROBtoPLC.User.Cycle.DO263_RingScanReach;
   END_TRANSITION
   STEP ScanStart:   // S246, max time T#10S, warning time T#7S
          S1  S    "KeyenceSR1000Ctrl_804A1DB".ioAutoTrigger
   END_STEP
   TRANSITION Trans246 FROM ScanStart TO WaitScanCompletely   // T246
      := NOT "KeyenceSR1000Ctrl_804A1DB".sHMI.Status.Ready;
   END_TRANSITION
   STEP WaitScanCompletely:   // S247, max time T#10S, warning time T#7S
   END_STEP
   TRANSITION Trans247 FROM WaitScanCompletely TO CodeMove   // T247
      := "KeyenceSR1000Ctrl_804A1DB".sHMI.Status.Complete AND "KeyenceSR1000Ctrl_804A1DB".sHMI.Status.ReadOk;
   END_TRANSITION
   TRANSITION Trans248 FROM WaitScanCompletely TO PartNGStatus   // T248
      := "KeyenceSR1000Ctrl_804A1DB".sHMI.Status.Complete AND "KeyenceSR1000Ctrl_804A1DB".sHMI.Status.ReadNok;
   END_TRANSITION
   STEP CodeMove:   // S248, max time T#10S, warning time T#7S
              N    "AutoProcessData".F_Robot1Grip2.RingCode_1:="KeyenceSR1000Ctrl_804A1DB".sHMI.Status.CurrentCode
   END_STEP
   TRANSITION Trans249 FROM CodeMove TO PartOKStatus_1   // T249
      := TRUE;
   END_TRANSITION
   STEP PartOKStatus:   // S249, max time T#10S, warning time T#7S
              N    "AutoProcessData".F_Robot1Grip2.PartStatus:=199
   END_STEP
   TRANSITION Trans251 FROM PartOKStatus TO WaitRobotFinish_4   // T251
      := "AutoProcessData".F_Robot1Grip2.PartStatus = 199;
   END_TRANSITION
   STEP PartNGStatus:   // S251, max time T#10S, warning time T#7S
              N    "AutoProcessData".F_Robot1Grip2.PartStatus:=150
   END_STEP
   TRANSITION Trans252 FROM PartNGStatus TO WaitRobotFinish_4   // T252
      := "AutoProcessData".F_Robot1Grip2.PartStatus = 150;
   END_TRANSITION
   STEP PartOKStatus_1:   // S266, max time T#10S, warning time T#7S
              N    "AutoProcessData".F_Robot1Grip2.PartStatus:=110
   END_STEP
   TRANSITION Trans267 FROM PartOKStatus_1 TO "MES Online  offline?"   // T267
      := "AutoProcessData".F_Robot1Grip2.PartStatus = 110;
   END_TRANSITION
   STEP "MES Online  offline?":   // S384, max time T#10S, warning time T#7S
   END_STEP
   TRANSITION Offline FROM "MES Online  offline?" TO PartOKStatus   // T698
      := "Station_Sys".Cmd.OnOffLine;
   END_TRANSITION
   TRANSITION Trans702 FROM "MES Online  offline?" TO WaitRobotFinish_4   // T702
      := NOT "Station_Sys".Cmd.OnOffLine;
   END_TRANSITION

   // sequencer 9
   STEP PressShaftPutProcess:   // S500, max time T#10S, warning time T#7S
   END_STEP
   TRANSITION Trans500 FROM PressShaftPutProcess TO StartRobotPressShaftPut   // T500
      := TRUE;
   END_TRANSITION
   STEP DataMove_2:   // S257, max time T#10S, warning time T#7S
          S1  N    "AutoProcessData".B_Press1:="AutoProcessData".F_Robot1Grip1
          S1  N    "AutoProcessData".F_Robot1Grip1:="AutoProcessData".ClearData
   END_STEP
   TRANSITION Trans258 FROM DataMove_2 TO WaitRobotFinish_5   // T258
      := #DataMove_2.T > t#100MS;
   END_TRANSITION
   STEP StartRobotPressShaftPut:   // S358, max time T#10S, warning time T#7S
              N    "KukaRobot1_CtrlDB".sPLCtoROB.User.Cycle.DI273_PressShaftPutReq
   END_STEP
   TRANSITION Trans646 FROM StartRobotPressShaftPut TO WaitRobotGripStatus   // T663
      := "KukaRobot1_CtrlDB".sROBtoPLC.User.Cycle.DO273_PressShaftPutInside AND NOT "KukaRobot1_CtrlDB".sROBtoPLC.User.Cycle.DO274_PressShaftPutFinish;
   END_TRANSITION
   STEP WaitRobotFinish_5:   // S359, max time T#10S, warning time T#7S
   END_STEP
   TRANSITION P13 FROM WaitRobotFinish_5 TO PressShaftPutProcessFinish   // T664
      := "KukaRobot1_CtrlDB".sROBtoPLC.User.Cycle.DO274_PressShaftPutFinish;
   END_TRANSITION
   STEP PressShaftPutProcessFinish:   // S549, max time T#10S, warning time T#7S
              S    #ioPM_Inface.ProcessComplete
              R    #ioPM_Inface.ProcessStart
              N    "AutoProcessData".F_Robot1Grip1.PartStatus:=0
   END_STEP
   TRANSITION Trans664 FROM PressShaftPutProcessFinish TO ProcessStart   // T549, jump
      := TRUE;
   END_TRANSITION
   STEP WaitRobotGripStatus:   // S360, max time T#10S, warning time T#7S
   END_STEP
   TRANSITION Trans665 FROM WaitRobotGripStatus TO DataMove_2   // T665
      := "KukaRobot1_CtrlDB".sROBtoPLC.User.Public.GO5_RobGrip1Status = 0;
   END_TRANSITION

   // sequencer 10
   STEP PressRingPutProcess:   // S550, max time T#10S, warning time T#7S
   END_STEP
   TRANSITION Trans550 FROM PressRingPutProcess TO StartRobotPressRingPut   // T550
      := TRUE;
   END_TRANSITION
   STEP DataMove_3:   // S260, max time T#10S, warning time T#7S
          S1  N    "AutoProcessData".B_Press1.RingCode_1:="AutoProcessData".F_Robot1Grip2.RingCode_1
          S1  N    "AutoProcessData".F_Robot1Grip2:="AutoProcessData".ClearData
              N    "AutoProcessData".B_Press1.PartStatus:=220
   END_STEP
   TRANSITION Trans261 FROM DataMove_3 TO WaitRobotFinish_6   // T261
      := (#DataMove_3.T > t#100MS) AND ("AutoProcessData".B_Press1.PartStatus = 220);
   END_TRANSITION
   STEP StartRobotPressRingPut:   // S361, max time T#10S, warning time T#7S
              N    "KukaRobot1_CtrlDB".sPLCtoROB.User.Cycle.DI277_PressRingPutReq
   END_STEP
   TRANSITION Trans647 FROM StartRobotPressRingPut TO WaitRobotGripStatus_1   // T666
      := "KukaRobot1_CtrlDB".sROBtoPLC.User.Cycle.DO277_PressRingPutInside AND NOT "KukaRobot1_CtrlDB".sROBtoPLC.User.Cycle.DO278_PressRingPutFinish;
   END_TRANSITION
   STEP WaitRobotFinish_6:   // S362, max time T#10S, warning time T#7S
   END_STEP
   TRANSITION P14 FROM WaitRobotFinish_6 TO PressRingPutProcessFinish   // T667
      := "KukaRobot1_CtrlDB".sROBtoPLC.User.Cycle.DO278_PressRingPutFinish;
   END_TRANSITION
   STEP PressRingPutProcessFinish:   // S599, max time T#10S, warning time T#7S
              S    #ioPM_Inface.ProcessComplete
              R    #ioPM_Inface.ProcessStart
   END_STEP
   TRANSITION Trans666 FROM PressRingPutProcessFinish TO ProcessStart   // T599, jump
      := TRUE;
   END_TRANSITION
   STEP WaitRobotGripStatus_1:   // S363, max time T#10S, warning time T#7S
   END_STEP
   TRANSITION Trans667 FROM WaitRobotGripStatus_1 TO DataMove_3   // T668
      := "KukaRobot1_CtrlDB".sROBtoPLC.User.Public.GO6_RobGrip2Status = 0;
   END_TRANSITION

   // sequencer 11
   STEP PressPickProcess:   // S600, max time T#10S, warning time T#7S
   END_STEP
   TRANSITION Trans600 FROM PressPickProcess TO StartRobotPressPick   // T600
      := TRUE;
   END_TRANSITION
   STEP DataMove_4:   // S262, max time T#10S, warning time T#7S
          S1  N    "AutoProcessData".F_Robot1Grip1:="AutoProcessData".B_Press1
          S1  N    "AutoProcessData".B_Press1:="AutoProcessData".ClearData
   END_STEP
   TRANSITION Trans263 FROM DataMove_4 TO WaitRobotFinish_7   // T263
      := #DataMove_4.T > t#100MS;
   END_TRANSITION
   STEP StartRobotPressPick:   // S364, max time T#10S, warning time T#7S
              N    "KukaRobot1_CtrlDB".sPLCtoROB.User.Cycle.DI281_PressPickShaftReq
   END_STEP
   TRANSITION Trans648 FROM StartRobotPressPick TO WaitRobotGripStatus_2   // T669
      := "KukaRobot1_CtrlDB".sROBtoPLC.User.Cycle.DO281_PressPickInside AND NOT "KukaRobot1_CtrlDB".sROBtoPLC.User.Cycle.DO282_PressPickFinish;
   END_TRANSITION
   STEP WaitRobotFinish_7:   // S365, max time T#10S, warning time T#7S
   END_STEP
   TRANSITION P15 FROM WaitRobotFinish_7 TO PressPickProcessFinish_   // T670
      := "KukaRobot1_CtrlDB".sROBtoPLC.User.Cycle.DO282_PressPickFinish;
   END_TRANSITION
   STEP PressPickProcessFinish_:   // S649, max time T#10S, warning time T#7S
              S    #ioPM_Inface.ProcessComplete
              R    #ioPM_Inface.ProcessStart
   END_STEP
   TRANSITION Trans668 FROM PressPickProcessFinish_ TO ProcessStart   // T649, jump
      := TRUE;
   END_TRANSITION
   STEP WaitRobotGripStatus_2:   // S366, max time T#10S, warning time T#7S
   END_STEP
   TRANSITION Trans669 FROM WaitRobotGripStatus_2 TO DataMove_4   // T671
      := "KukaRobot1_CtrlDB".sROBtoPLC.User.Public.GO5_RobGrip1Status <> 0;
   END_TRANSITION

   // sequencer 12
   STEP GluePutProcess:   // S650, max time T#10S, warning time T#7S
   END_STEP
   TRANSITION Trans674 FROM GluePutProcess TO StartRobotGluePut   // T650
      := TRUE;
   END_TRANSITION
   STEP DataMove_5:   // S264, max time T#10S, warning time T#7S
          S1  N    "AutoProcessData".C_Glue:="AutoProcessData".F_Robot1Grip1
          S1  N    "AutoProcessData".F_Robot1Grip1:="AutoProcessData".ClearData
   END_STEP
   TRANSITION Trans265 FROM DataMove_5 TO WaitRobotFinish_8   // T265
      := #DataMove_5.T > t#100MS;
   END_TRANSITION
   STEP StartRobotGluePut:   // S367, max time T#10S, warning time T#7S
              N    "KukaRobot1_CtrlDB".sPLCtoROB.User.Cycle.DI289_GluePutReq
   END_STEP
   TRANSITION Trans650 FROM StartRobotGluePut TO WaitRobotGripStatus_3   // T676
      := "KukaRobot1_CtrlDB".sROBtoPLC.User.Cycle.DO289_GluePutInside AND NOT "KukaRobot1_CtrlDB".sROBtoPLC.User.Cycle.DO290_GluePutFinish;
   END_TRANSITION
   STEP WaitRobotFinish_8:   // S368, max time T#10S, warning time T#7S
   END_STEP
   TRANSITION P16 FROM WaitRobotFinish_8 TO GluePutProcessFinish   // T677
      := "KukaRobot1_CtrlDB".sROBtoPLC.User.Cycle.DO290_GluePutFinish;
   END_TRANSITION
   STEP GluePutProcessFinish:   // S699, max time T#10S, warning time T#7S
              S    #ioPM_Inface.ProcessComplete
              R    #ioPM_Inface.ProcessStart
              N    "Robot_DB".Robot_1.SpeedCount:="Robot_DB".Robot_1.SpeedCount+1
   END_STEP
   TRANSITION Trans670 FROM GluePutProcessFinish TO ProcessStart   // T699, jump
      := TRUE;
   END_TRANSITION
   STEP WaitRobotGripStatus_3:   // S369, max time T#10S, warning time T#7S
   END_STEP
   TRANSITION Trans671 FROM WaitRobotGripStatus_3 TO DataMove_5   // T679
      := "KukaRobot1_CtrlDB".sROBtoPLC.User.Public.GO5_RobGrip1Status = 0;
   END_TRANSITION

   // sequencer 13
   STEP "NG PutProcess":   // S700, max time T#10S, warning time T#7S
   END_STEP
   TRANSITION Trans700 FROM "NG PutProcess" TO StartRobotNGPut   // T700
      := TRUE;
   END_TRANSITION
   STEP StartRobotNGPut:   // S370, max time T#10S, warning time T#7S
              N    "KukaRobot1_CtrlDB".sPLCtoROB.User.Cycle.DI265_LoadPressNGReq1
   END_STEP
   TRANSITION Trans651 FROM StartRobotNGPut TO WaitRobotGripStatus_4   // T680
      := "KukaRobot1_CtrlDB".sROBtoPLC.User.Cycle.DO265_LoadNGInside AND NOT "KukaRobot1_CtrlDB".sROBtoPLC.User.Cycle.DO266_LoadNGFinish;
   END_TRANSITION
   STEP WaitRobotFinish_9:   // S371, max time T#10S, warning time T#7S
   END_STEP
   TRANSITION P17 FROM WaitRobotFinish_9 TO "NG1 PutProcessFinish"   // T681
      := "KukaRobot1_CtrlDB".sROBtoPLC.User.Cycle.DO266_LoadNGFinish;
   END_TRANSITION
   STEP "NG1 PutProcessFinish":   // S749, max time T#10S, warning time T#7S
              S    #ioPM_Inface.ProcessComplete
              R    #ioPM_Inface.ProcessStart
   END_STEP
   TRANSITION Trans673 FROM "NG1 PutProcessFinish" TO ProcessStart   // T749, jump
      := TRUE;
   END_TRANSITION
   STEP WaitRobotGripStatus_4:   // S372, max time T#10S, warning time T#7S
   END_STEP
   TRANSITION Trans678 FROM WaitRobotGripStatus_4 TO "Data Clear_7"   // T682
      := "KukaRobot1_CtrlDB".sROBtoPLC.User.Public.GO5_RobGrip1Status = 0;
   END_TRANSITION
   STEP "Data Clear_7":   // S267, max time T#10S, warning time T#7S
      // CJ - check why
          S1  N    "AutoProcessData".F_Robot1Grip1:="AutoProcessData".ClearData
   END_STEP
   TRANSITION Trans268 FROM "Data Clear_7" TO WaitRobotFinish_9   // T268
      := TRUE;
   END_TRANSITION

   // sequencer 14
   STEP "Data Clear_8":   // S268, max time T#10S, warning time T#7S
          S1  N    "AutoProcessData".F_Robot1Grip1:="AutoProcessData".ClearData
   END_STEP
   TRANSITION Trans269 FROM "Data Clear_8" TO WaitRobotFinish_10   // T269
      := TRUE;
   END_TRANSITION
   STEP "NG 2 PutProcess":   // S750, max time T#10S, warning time T#7S
   END_STEP
   TRANSITION Trans701 FROM "NG 2 PutProcess" TO StartRobotNG2Put_1   // T750
      := TRUE;
   END_TRANSITION
   STEP StartRobotNG2Put_1:   // S373, max time T#10S, warning time T#7S
              N    "KukaRobot1_CtrlDB".sPLCtoROB.User.Cycle.DI266_LoadShaftScanNGReq2
   END_STEP
   TRANSITION Trans652 FROM StartRobotNG2Put_1 TO WaitRobotGripStatus_5   // T685
      := "KukaRobot1_CtrlDB".sROBtoPLC.User.Cycle.DO265_LoadNGInside AND NOT "KukaRobot1_CtrlDB".sROBtoPLC.User.Cycle.DO266_LoadNGFinish;
   END_TRANSITION
   STEP WaitRobotFinish_10:   // S374, max time T#10S, warning time T#7S
   END_STEP
   TRANSITION P18 FROM WaitRobotFinish_10 TO "NG2 PutProcessFinish"   // T686
      := "KukaRobot1_CtrlDB".sROBtoPLC.User.Cycle.DO266_LoadNGFinish;
   END_TRANSITION
   STEP "NG2 PutProcessFinish":   // S799, max time T#10S, warning time T#7S
              S    #ioPM_Inface.ProcessComplete
              R    #ioPM_Inface.ProcessStart
   END_STEP
   TRANSITION Trans680 FROM "NG2 PutProcessFinish" TO ProcessStart   // T799, jump
      := TRUE;
   END_TRANSITION
   STEP WaitRobotGripStatus_5:   // S375, max time T#10S, warning time T#7S
   END_STEP
   TRANSITION Trans681 FROM WaitRobotGripStatus_5 TO "Data Clear_8"   // T687
      := "KukaRobot1_CtrlDB".sROBtoPLC.User.Public.GO5_RobGrip1Status = 0;
   END_TRANSITION

   // sequencer 15
   STEP "NG 3 PutProcess":   // S800, max time T#10S, warning time T#7S
   END_STEP
   TRANSITION Trans752 FROM "NG 3 PutProcess" TO StartRobotNG3Put   // T800
      := TRUE;
   END_TRANSITION
   STEP "Data Clear_9":   // S269, max time T#10S, warning time T#7S
              N    "AutoProcessData".F_Robot1Grip2:="AutoProcessData".ClearData
   END_STEP
   TRANSITION Trans270 FROM "Data Clear_9" TO WaitRobotFinish_11   // T270
      := TRUE;
   END_TRANSITION
   STEP StartRobotNG3Put:   // S376, max time T#10S, warning time T#7S
              N    "KukaRobot1_CtrlDB".sPLCtoROB.User.Cycle.DI267_LoadRingScanNGReq3
   END_STEP
   TRANSITION Trans653 FROM StartRobotNG3Put TO WaitRobotGripStatus_6   // T688
      := "KukaRobot1_CtrlDB".sROBtoPLC.User.Cycle.DO265_LoadNGInside AND NOT "KukaRobot1_CtrlDB".sROBtoPLC.User.Cycle.DO266_LoadNGFinish;
   END_TRANSITION
   STEP WaitRobotFinish_11:   // S377, max time T#10S, warning time T#7S
   END_STEP
   TRANSITION P19 FROM WaitRobotFinish_11 TO "NG3 PutProcessFinish"   // T689
      := "KukaRobot1_CtrlDB".sROBtoPLC.User.Cycle.DO266_LoadNGFinish;
   END_TRANSITION
   STEP "NG3 PutProcessFinish":   // S849, max time T#10S, warning time T#7S
              S    #ioPM_Inface.ProcessComplete
              R    #ioPM_Inface.ProcessStart
   END_STEP
   TRANSITION Trans682 FROM "NG3 PutProcessFinish" TO ProcessStart   // T849, jump
      := TRUE;
   END_TRANSITION
   STEP WaitRobotGripStatus_6:   // S378, max time T#10S, warning time T#7S
   END_STEP
   TRANSITION Trans683 FROM WaitRobotGripStatus_6 TO "Data Clear_9"   // T690
      := "KukaRobot1_CtrlDB".sROBtoPLC.User.Public.GO6_RobGrip2Status = 0;
   END_TRANSITION

   // sequencer 16
   STEP "Maintenance Pos":   // S850, max time T#10S, warning time T#7S
   END_STEP
   TRANSITION Trans704 FROM "Maintenance Pos" TO ReqRobotToMantenPos   // T850
      := "KukaRobot2_CtrlDB".sROBtoPLC.User.Cycle.DO298_MaintainFinish OR "KukaRobot2_CtrlDB".sROBtoPLC.Sys.SO.IN_HOME;
   END_TRANSITION
   STEP ReqRobotToMantenPos:   // S701, max time T#10S, warning time T#7S
              N    "KukaRobot1_CtrlDB".sPLCtoROB.User.Cycle.DI297_MaintainRequest
   END_STEP
   TRANSITION Trans705 FROM ReqRobotToMantenPos TO WaitR1MaintenPosFinsh   // T703
      := "KukaRobot1_CtrlDB".sROBtoPLC.User.Cycle.DO297_MaintainInside AND NOT "KukaRobot1_CtrlDB".sROBtoPLC.User.Cycle.DO298_MaintainFinish;
   END_TRANSITION
   STEP WaitR1MaintenPosFinsh:   // S702, max time T#10S, warning time T#7S
              R    "AutoProcessControl".Robot_1.MaintenanceRequest
   END_STEP
   TRANSITION Trans706 FROM WaitR1MaintenPosFinsh TO WaitRobotHomeRequest   // T704
      := NOT "KukaRobot1_CtrlDB".sROBtoPLC.User.Cycle.DO297_MaintainInside AND "KukaRobot1_CtrlDB".sROBtoPLC.User.Cycle.DO298_MaintainFinish AND NOT "AutoProcessControl".Robot_1.MaintenanceRequest AND NOT "ChangeOver_DB".Robot_1.Req_RobotToMaintenancePos;
   END_TRANSITION
   STEP WaitRobotHomeRequest:   // S703, max time T#10S, warning time T#7S
          S1  R    "ChangeOver_DB".Robot_1.MaintenancePosReqSelFlag
   END_STEP
   TRANSITION Trans707 FROM WaitRobotHomeRequest TO ReqRobotToHomePos   // T705
      := "ChangeOver_DB".Robot_1.HMI_MaintenanceHomeReq AND NOT "KukaRobot1_CtrlDB".sROBtoPLC.User.Cycle.DO300_HomeInside AND ("KukaRobot2_CtrlDB".sROBtoPLC.User.Cycle.DO298_MaintainFinish OR "KukaRobot2_CtrlDB".sROBtoPLC.Sys.SO.IN_HOME);
   END_TRANSITION
   STEP ReqRobotToHomePos:   // S704, max time T#10S, warning time T#7S
              N    "KukaRobot1_CtrlDB".sPLCtoROB.User.Cycle.DI300_HomeRequest
   END_STEP
   TRANSITION Trans708 FROM ReqRobotToHomePos TO WaitR1HomePosFinsh_1   // T706
      := "KukaRobot1_CtrlDB".sROBtoPLC.User.Cycle.DO300_HomeInside AND NOT "KukaRobot1_CtrlDB".sROBtoPLC.User.Cycle.DO301_HomeFinish;
   END_TRANSITION
   STEP WaitR1HomePosFinsh_1:   // S899, max time T#10S, warning time T#7S
   END_STEP
   TRANSITION Trans709 FROM WaitR1HomePosFinsh_1 TO ProcessStart   // T899, jump
      := NOT "KukaRobot1_CtrlDB".sROBtoPLC.User.Cycle.DO300_HomeInside AND "KukaRobot1_CtrlDB".sROBtoPLC.User.Cycle.DO301_HomeFinish AND NOT "AutoProcessControl".Robot_1.HomeRequest;
   END_TRANSITION

   // sequencer 17
   STEP RobotTest:   // S900, max time T#10S, warning time T#7S
   END_STEP
   TRANSITION Trans134 FROM RobotTest TO MasteringTest_Req   // T134
      := TRUE;
   END_TRANSITION
   TRANSITION Trans137 FROM RobotTest TO BrakeTest_Req   // T137
      := TRUE;
   END_TRANSITION
   STEP MasteringTest_Req:   // S910, max time T#10S, warning time T#7S
              N    "KukaRobot1_CtrlDB".sPLCtoROB.User.Cycle.DI321
              N    "KukaRobot1_CtrlDB".sPLCtoROB.User.Safety.DI450
   END_STEP
   TRANSITION Trans136 FROM MasteringTest_Req TO WaitMasteringTestFinish   // T136
      := "KukaRobot1_CtrlDB".sROBtoPLC.User.Safety.DO462;
   END_TRANSITION
   STEP BrakeTest_Req:   // S920, max time T#10S, warning time T#7S
              N    "KukaRobot1_CtrlDB".sPLCtoROB.User.Cycle.DI329
              N    "KukaRobot1_CtrlDB".sPLCtoROB.User.Safety.DI451
   END_STEP
   TRANSITION Trans138 FROM BrakeTest_Req TO WaitBrakeTestFinish   // T138
      := "KukaRobot1_CtrlDB".sROBtoPLC.User.Safety.DO453;
   END_TRANSITION
   STEP WaitMasteringTestFinish:   // S911, max time T#10S, warning time T#7S
   END_STEP
   TRANSITION Trans139 FROM WaitMasteringTestFinish TO MasteringTestFinish   // T139
      := NOT "KukaRobot1_CtrlDB".sROBtoPLC.User.Safety.DO460 AND NOT "KukaRobot1_CtrlDB".sROBtoPLC.User.Safety.DO462 AND "KukaRobot1_CtrlDB".sROBtoPLC.User.Safety.DO461;
   END_TRANSITION
   STEP WaitBrakeTestFinish:   // S921, max time T#10S, warning time T#7S
   END_STEP
   TRANSITION Trans141 FROM WaitBrakeTestFinish TO BrakeTestFinish   // T141
      := NOT "KukaRobot1_CtrlDB".sROBtoPLC.User.Safety.DO452 AND NOT "KukaRobot1_CtrlDB".sROBtoPLC.User.Safety.DO453 AND "KukaRobot1_CtrlDB".sROBtoPLC.User.Safety.DO454;
   END_TRANSITION
   STEP MasteringTestFinish:   // S919, max time T#10S, warning time T#7S
              R    "Robot_DB".Robot_1.MasteringTest_Req
   END_STEP
   TRANSITION Trans142 FROM MasteringTestFinish TO ProcessStart   // T919, jump
      := NOT "Robot_DB".Robot_1.MasteringTest_Req;
   END_TRANSITION
   STEP BrakeTestFinish:   // S929, max time T#10S, warning time T#7S
              R    "Robot_DB".Robot_1.BrakeTest_Req
   END_STEP
   TRANSITION Trans995 FROM BrakeTestFinish TO ProcessStart   // T929, jump
      := NOT "Robot_DB".Robot_1.BrakeTest_Req;
   END_TRANSITION

   // permanent post-instructions
   NETWORK 1
      #ioPM_Inface.StepNum := #RT_DATA.S_DISPLAY;
   NETWORK 2
      IF #iSysInface.Reset THEN #AlarmID := 0; END_IF;
   NETWORK 3
      #TON[10].TON(IN := #工件放行中, PT := T#0.5S);
      IF #TON[10].Q THEN #工件放行中 := FALSE; END_IF;
END_FUNCTION_BLOCK

FUNCTION_BLOCK "ST10_Flow6_ToolCodeScan"   // FB1076, GRAPH
// stored: AcknowledgeErrorsRequired false, AutoNumber false, GraphVersion 6.0, InitialValuesAcquisition false, SetENOAutomatically false
   // inherited from GRAPH_BASE
   VAR_INPUT
      iSysInface : "RCS_SysComInterface_V1";
   END_VAR
   VAR_IN_OUT
      ioPM_Inface : "RCS_PMInterface_V1";
      ioStatus : Int;
   END_VAR
   VAR
      sCtrlMode { S7_SetPoint := 'True'} : "SysFlowCtrlGraph";
      sUpdMES_Data : Bool;   // 更新MES数据
      工件放行中 : Bool;
      前站站号 { ExternalAccessible := 'False'; ExternalVisible := 'False'; ExternalWritable := 'False'} : UInt;
      本站站号 { ExternalAccessible := 'False'; ExternalVisible := 'False'; ExternalWritable := 'False'} : UInt;
      弹窗Temp : Array[1..10] of Int;
      AlarmID : Int;
      TON { S7_SetPoint := 'True'} : Array[0..10] of TON_TIME;
      TOF { S7_SetPoint := 'True'} : Array[0..10] of TOF_TIME;
      sUP { S7_SetPoint := 'True'} : Array[0..10] of Bool;
      更新RFID完成 : Bool;
   END_VAR
   VAR_TEMP
      Tempresult : USInt;
      本站站号乘10 : UInt;
   END_VAR
   // // TON[0] : 托盘流入1托盘到位传感器 / iA-Rotating product Check
   // // TON[1] : 托盘流入1托盘到位传感器
   // // TON[2] : 托盘流入1产品有无传感器
   // // TON[3] : 托盘流入1产品有无传感器
   // // TON[4] : 托盘流入1姿态检测光电2
   // // TON[5] : 托盘流入1姿态检测光电3
   // // TON[0].Q : 托盘流入1托盘到位 / iA-Rotating product Check
   // // TON[1].Q : 托盘流入1托盘无
   // // TON[2].Q : 托盘流入1有产品
   // // TON[3].Q : 托盘流入1无产品
   // // TON[4].Q : 托盘流入1姿态检测光电2
   // // TON[5].Q : 托盘流入1姿态检测光电3
   // // TOF[1] : iA-Rotating product Check
BEGIN
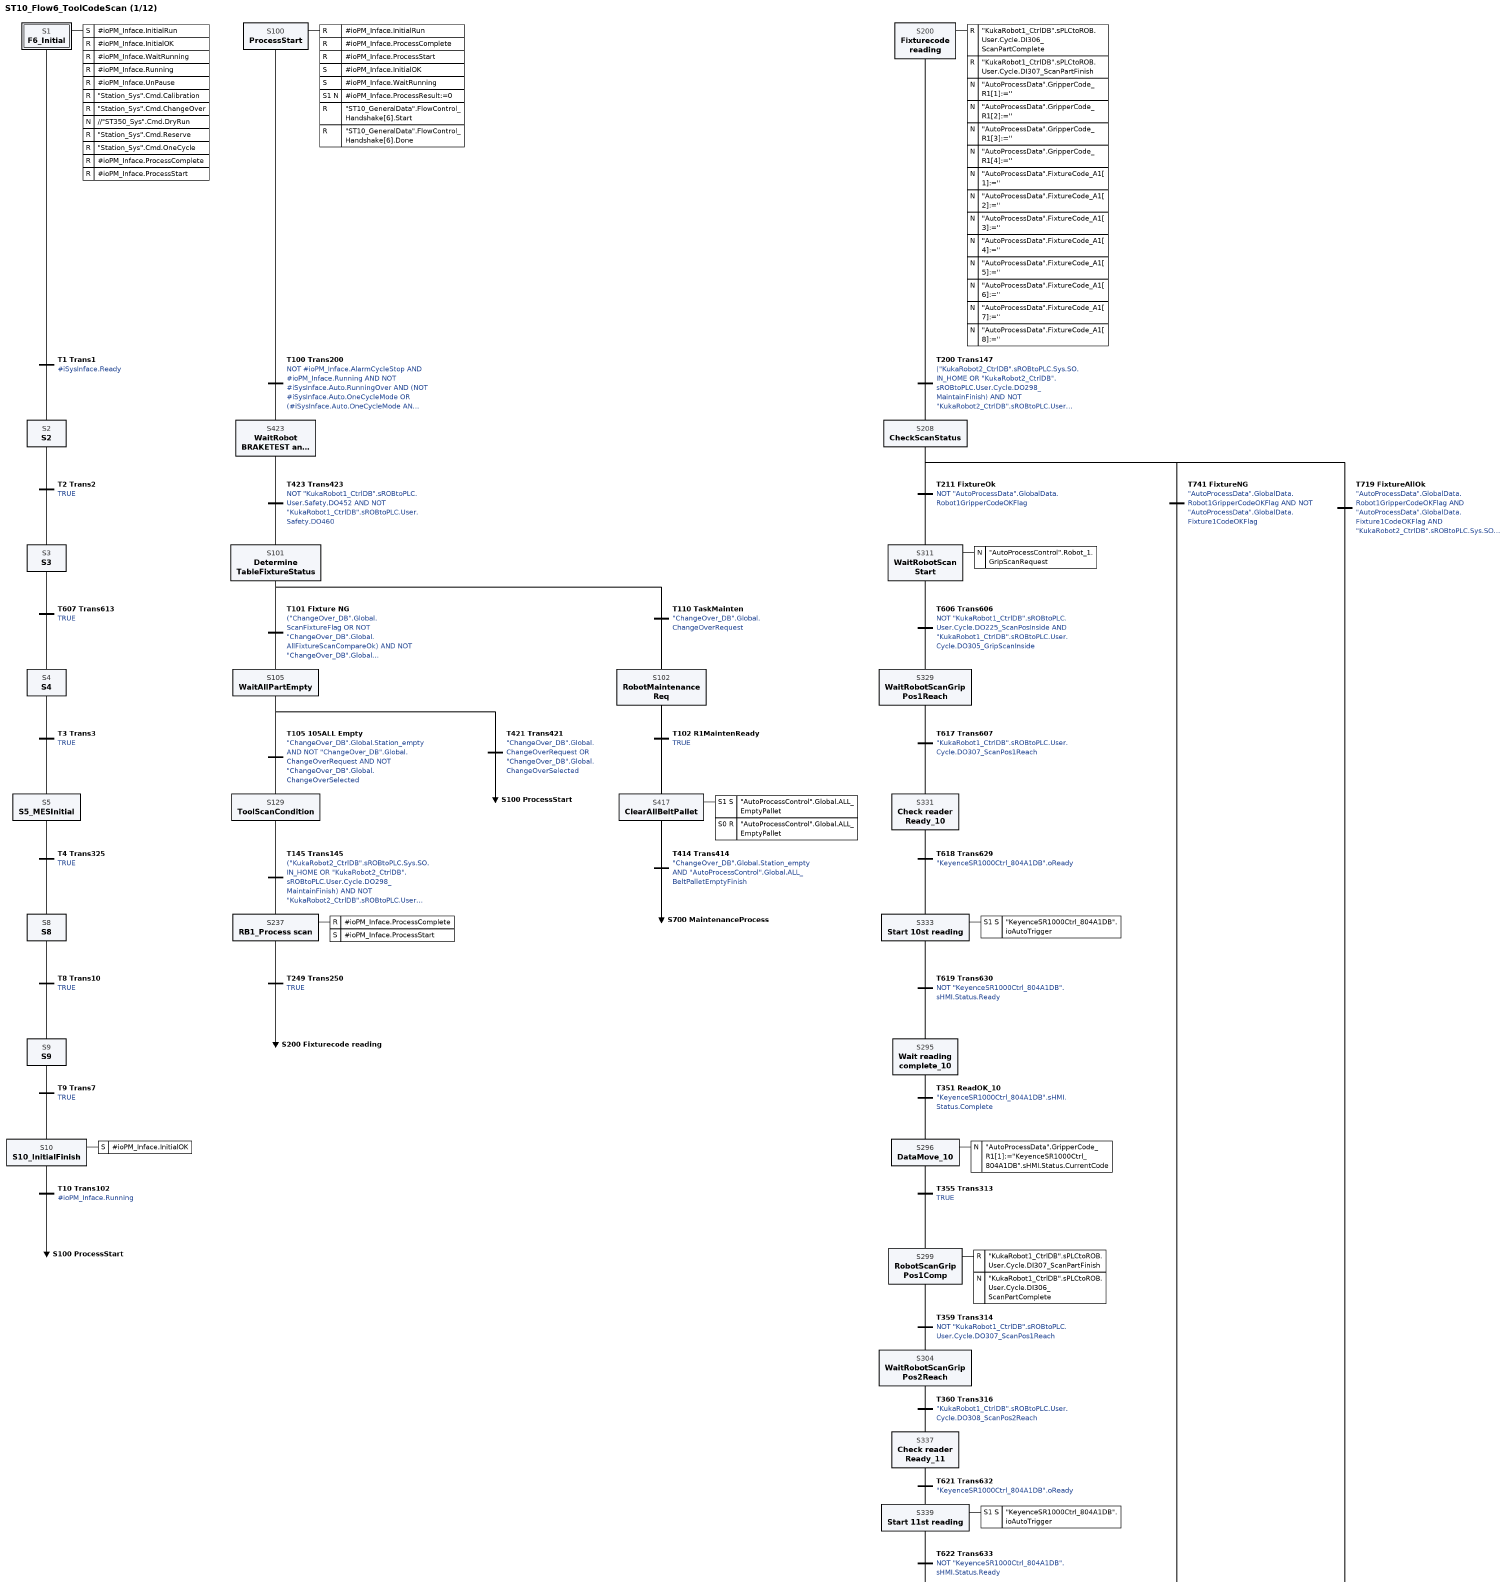
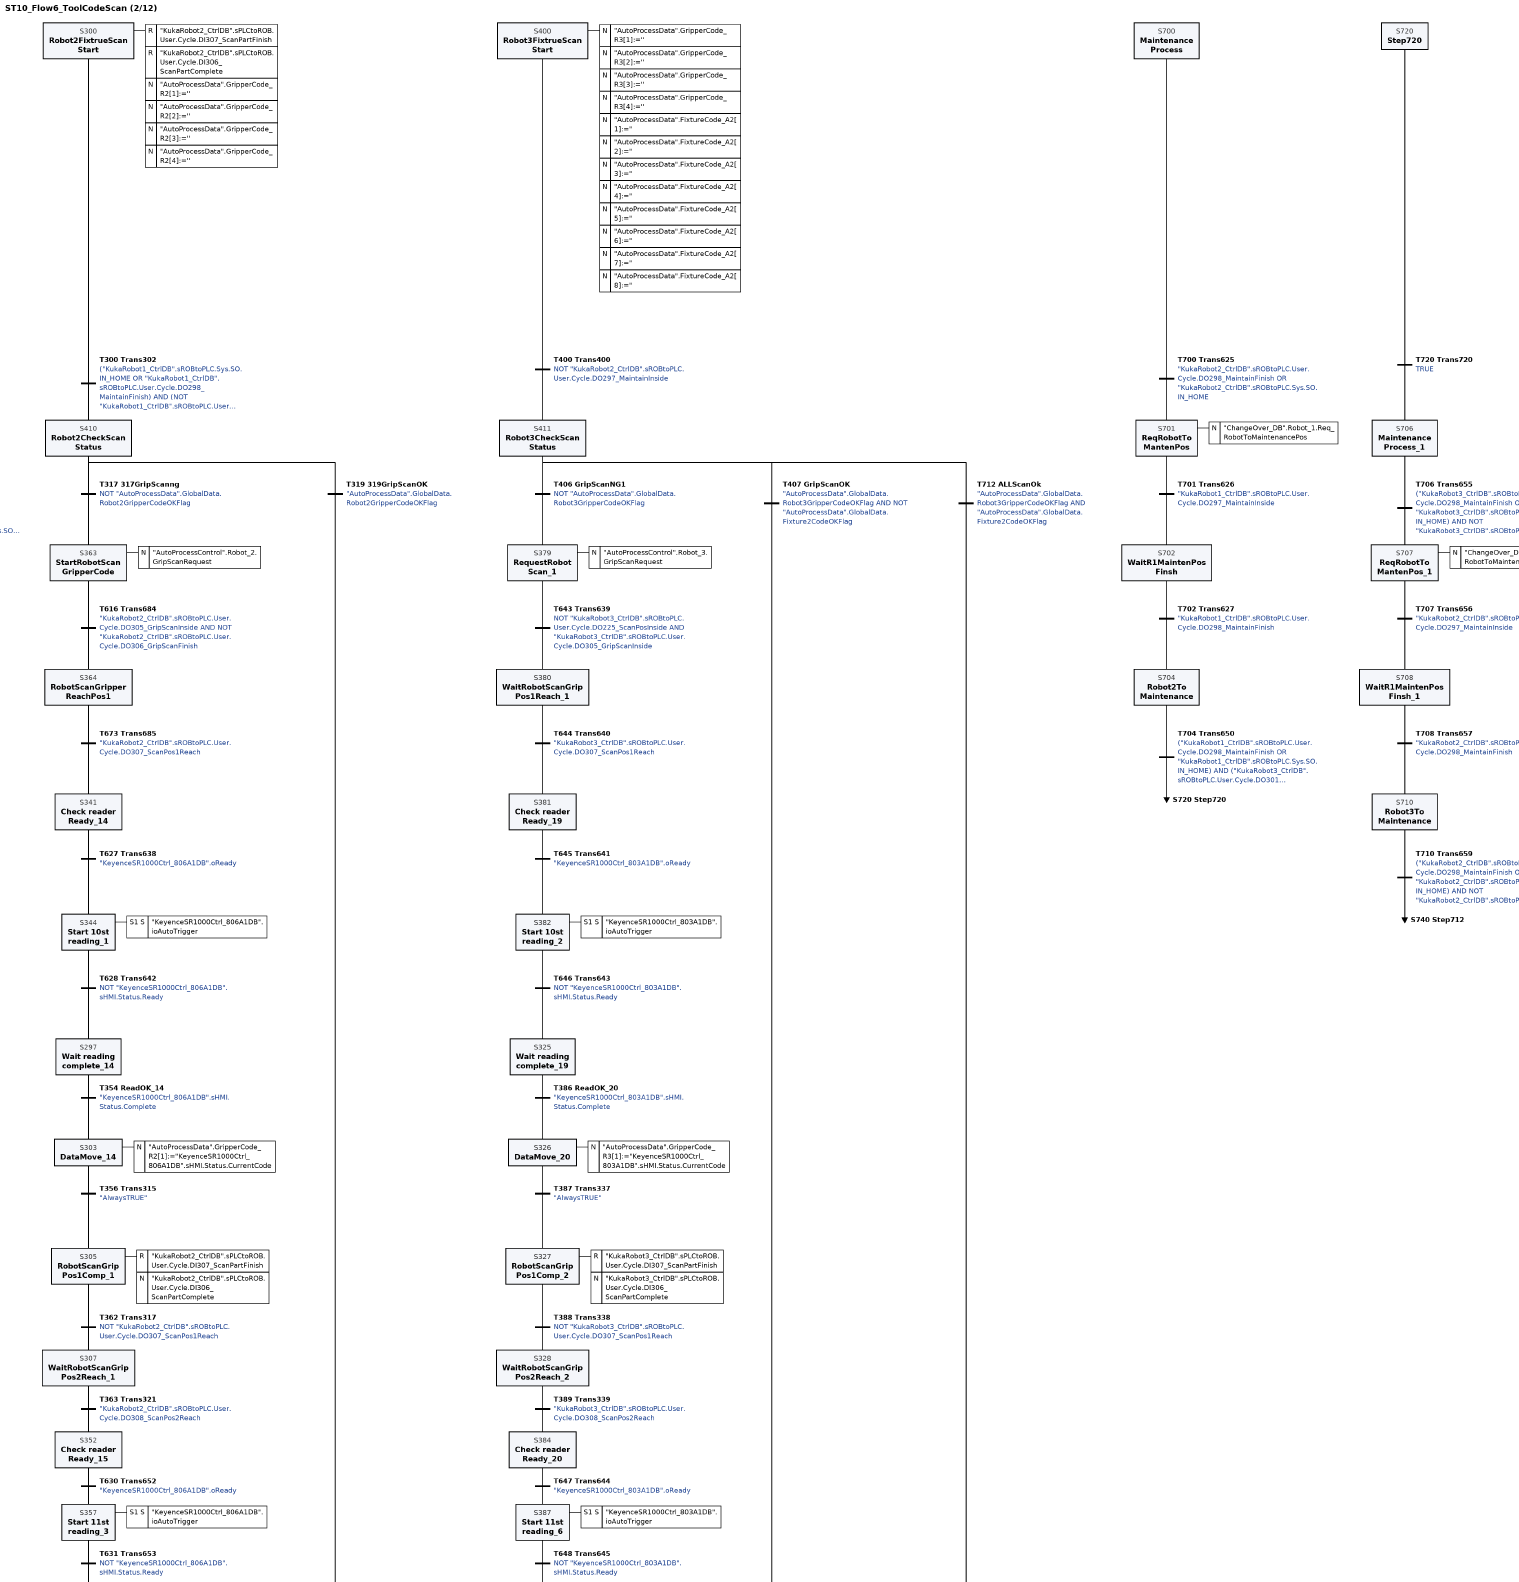
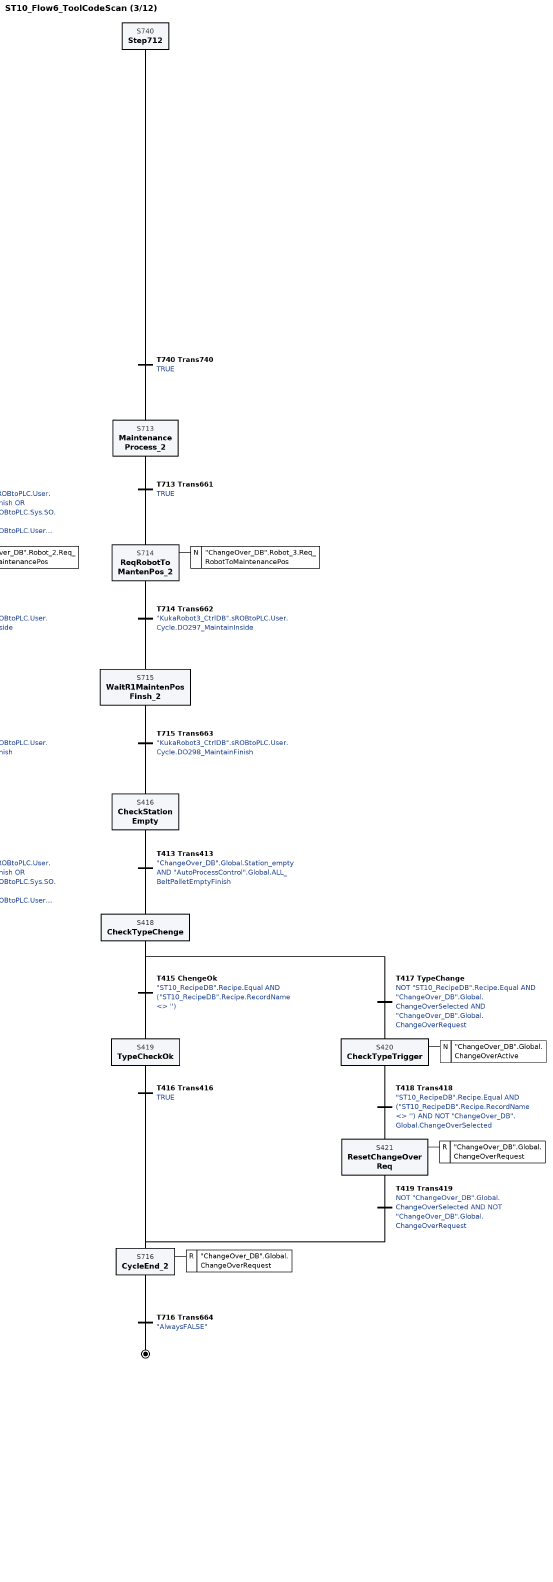
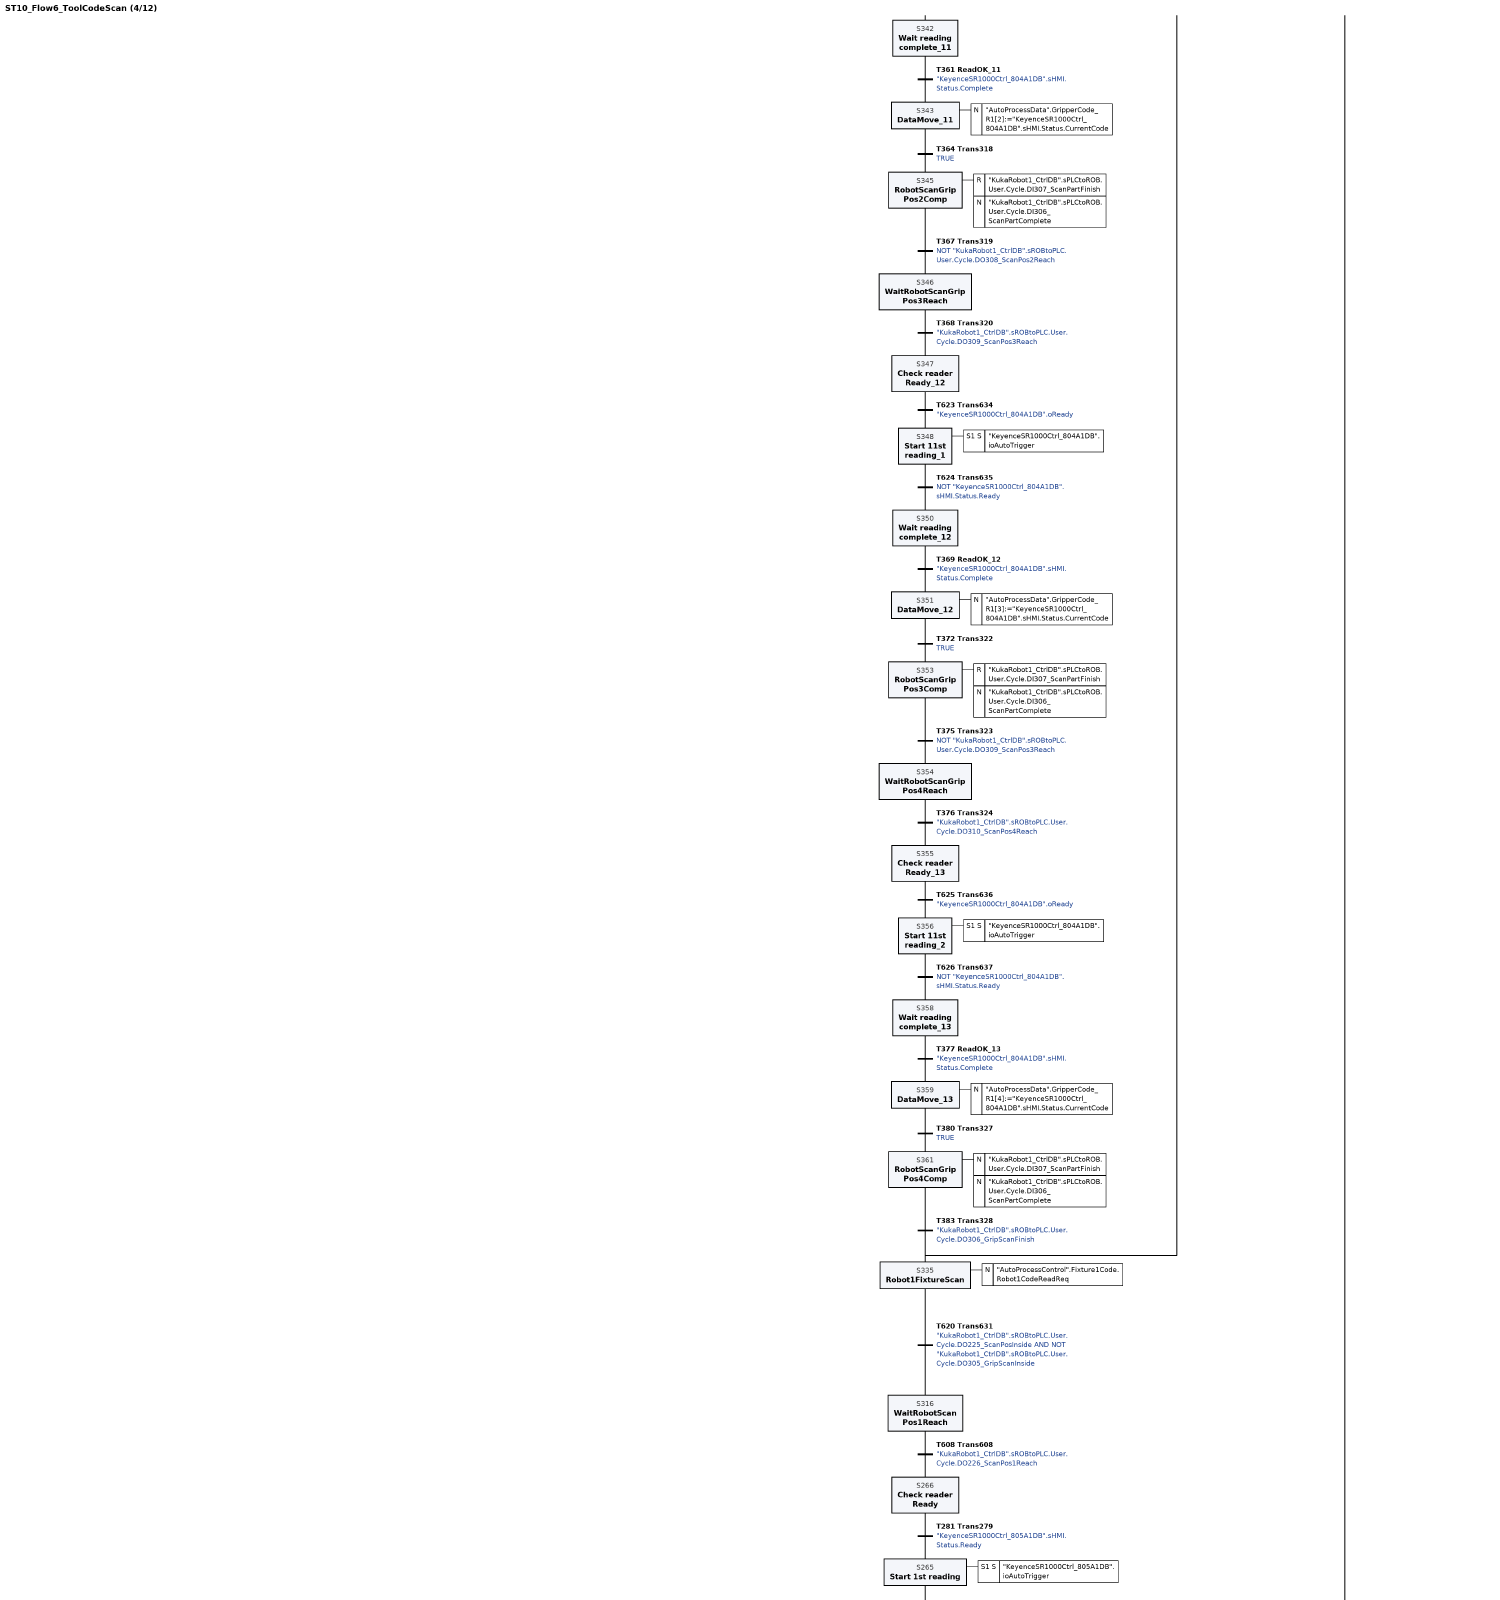
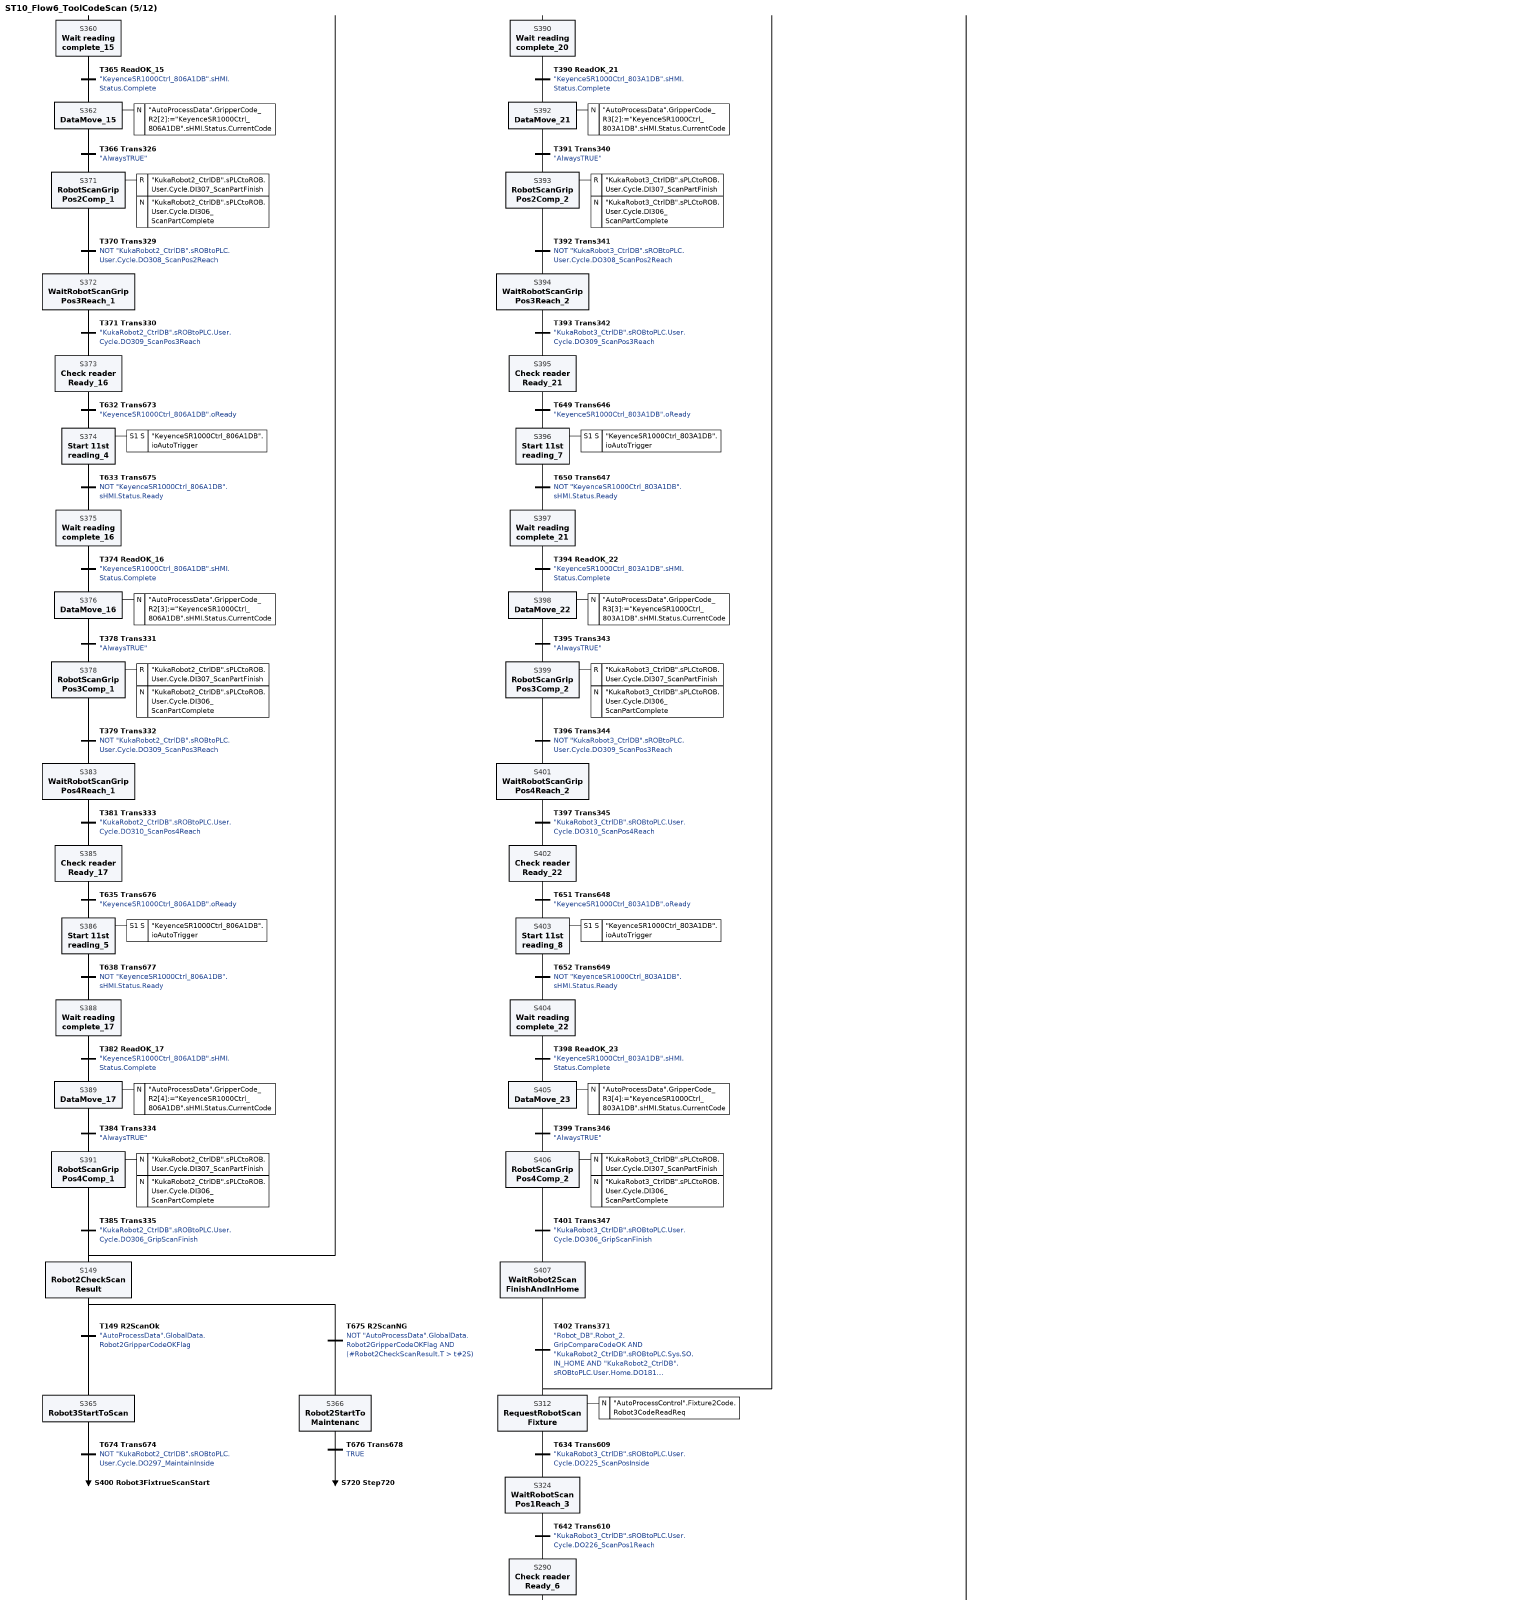
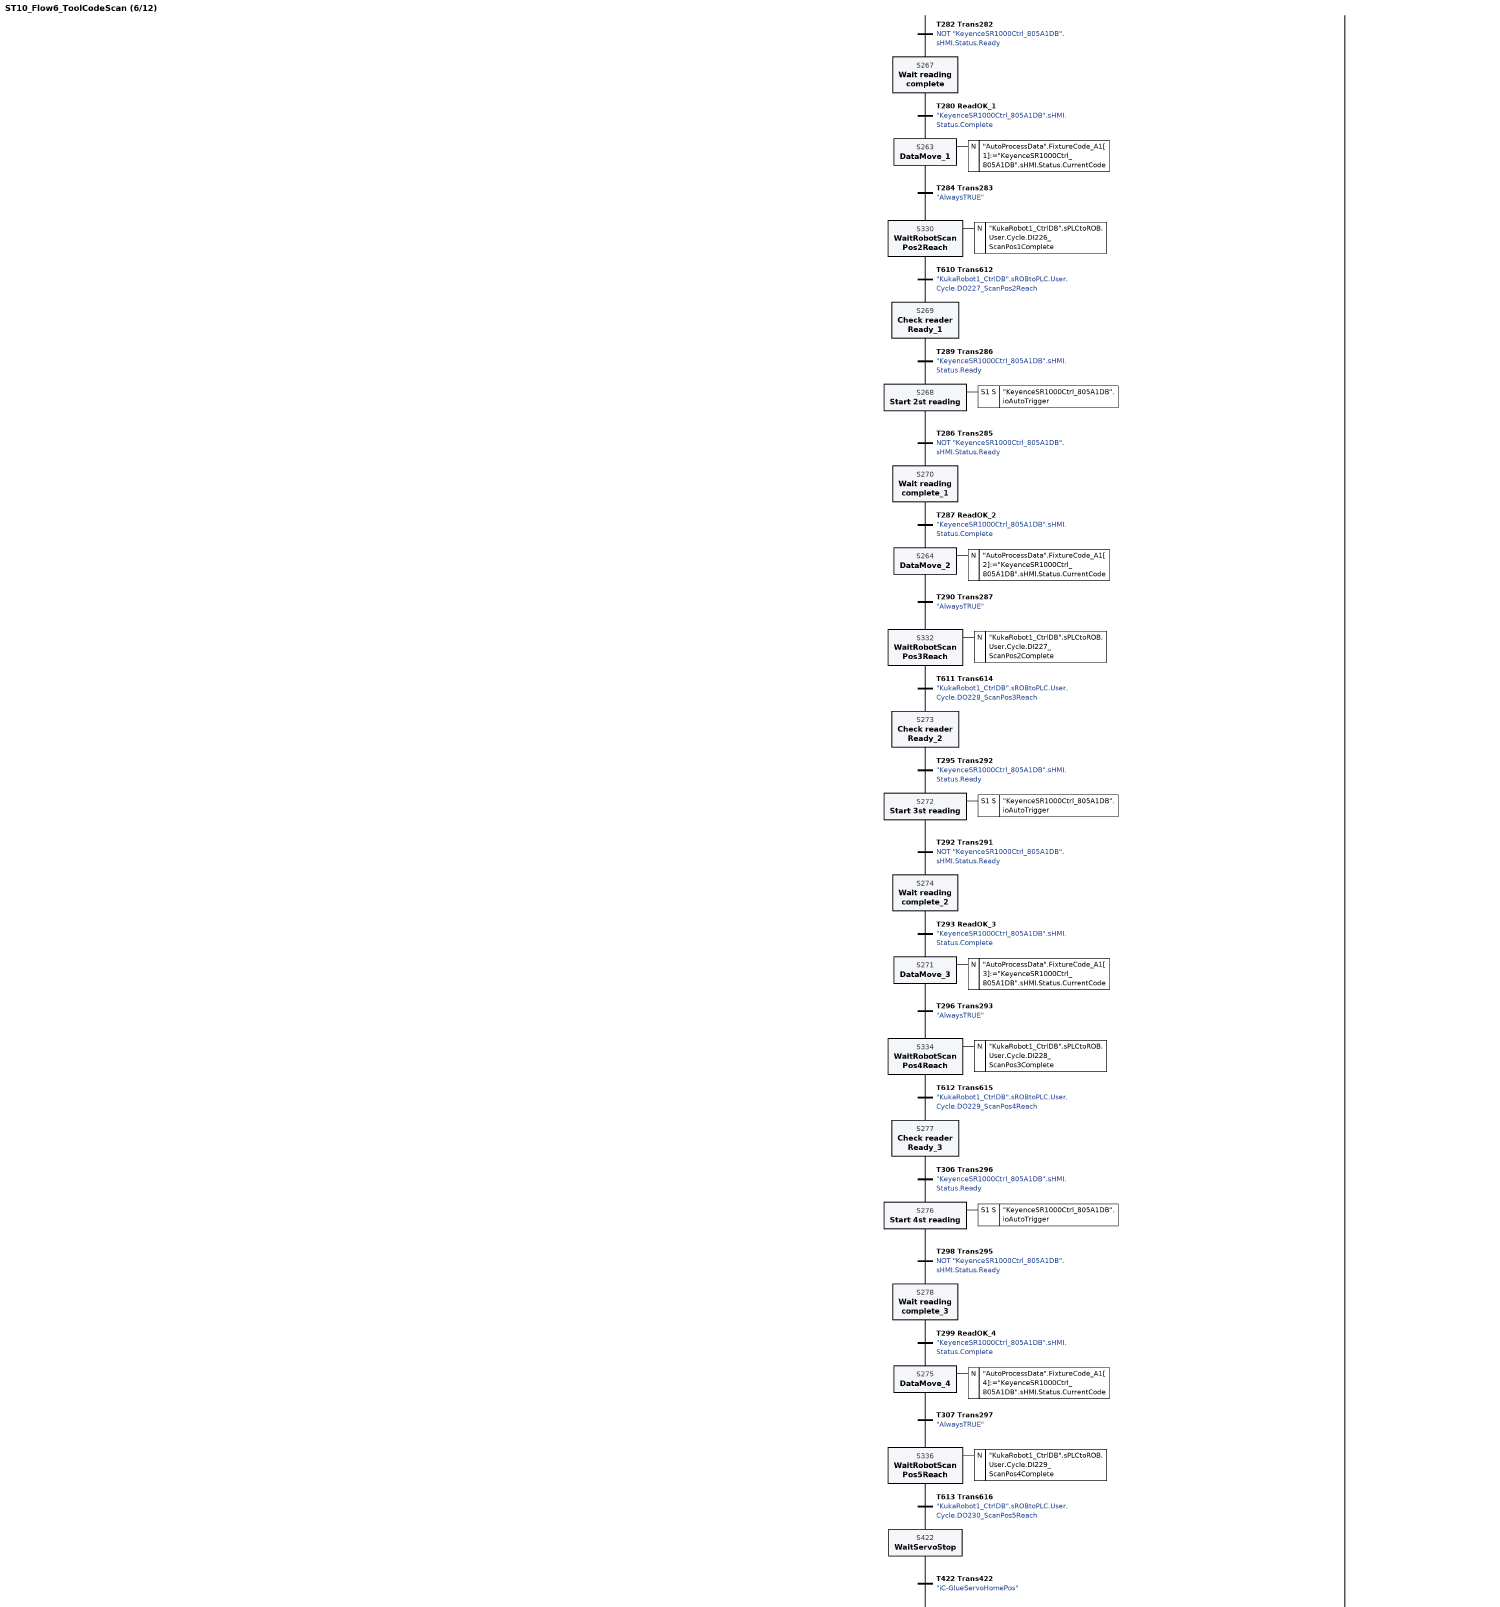
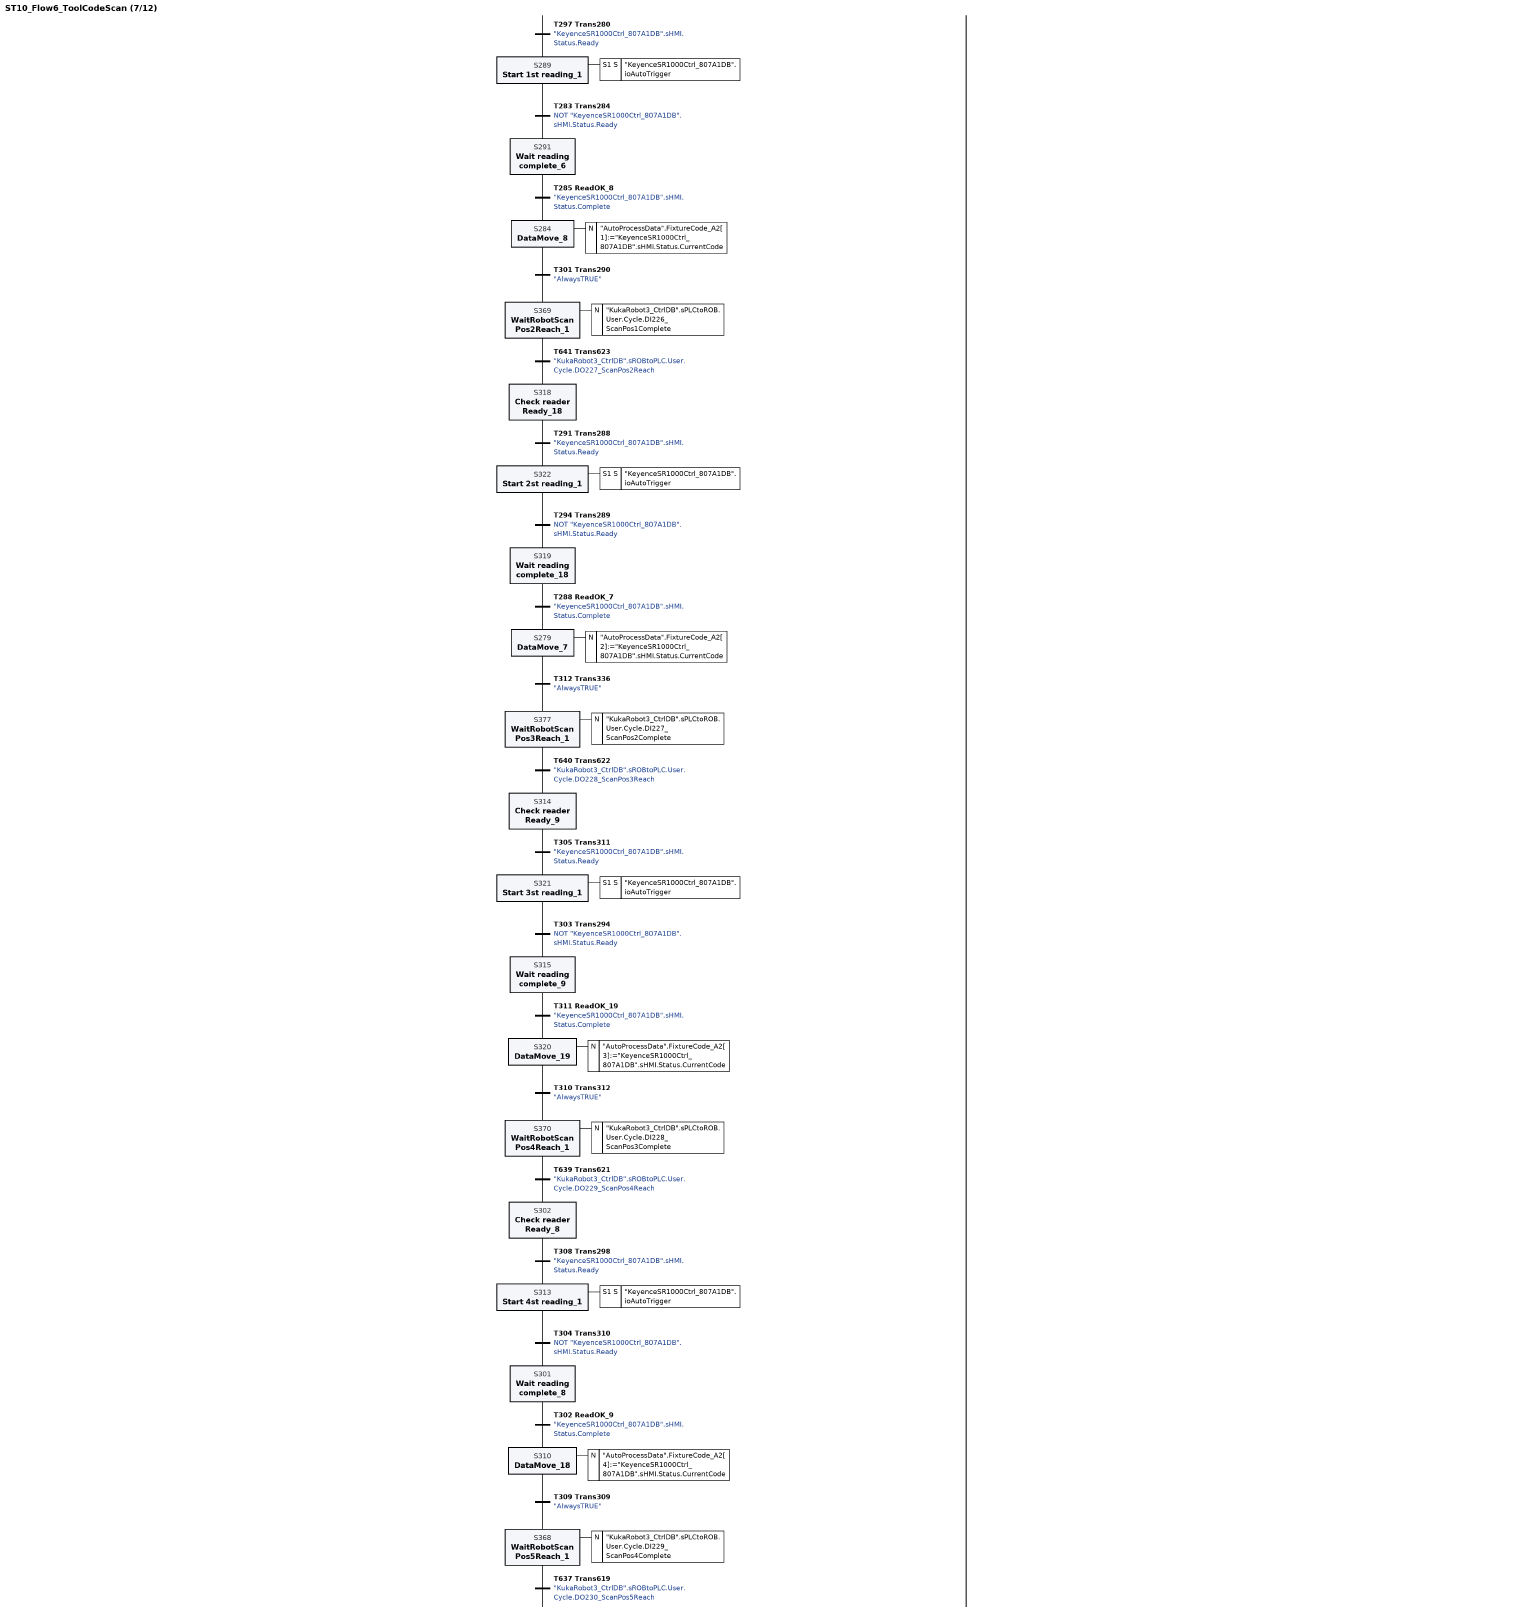
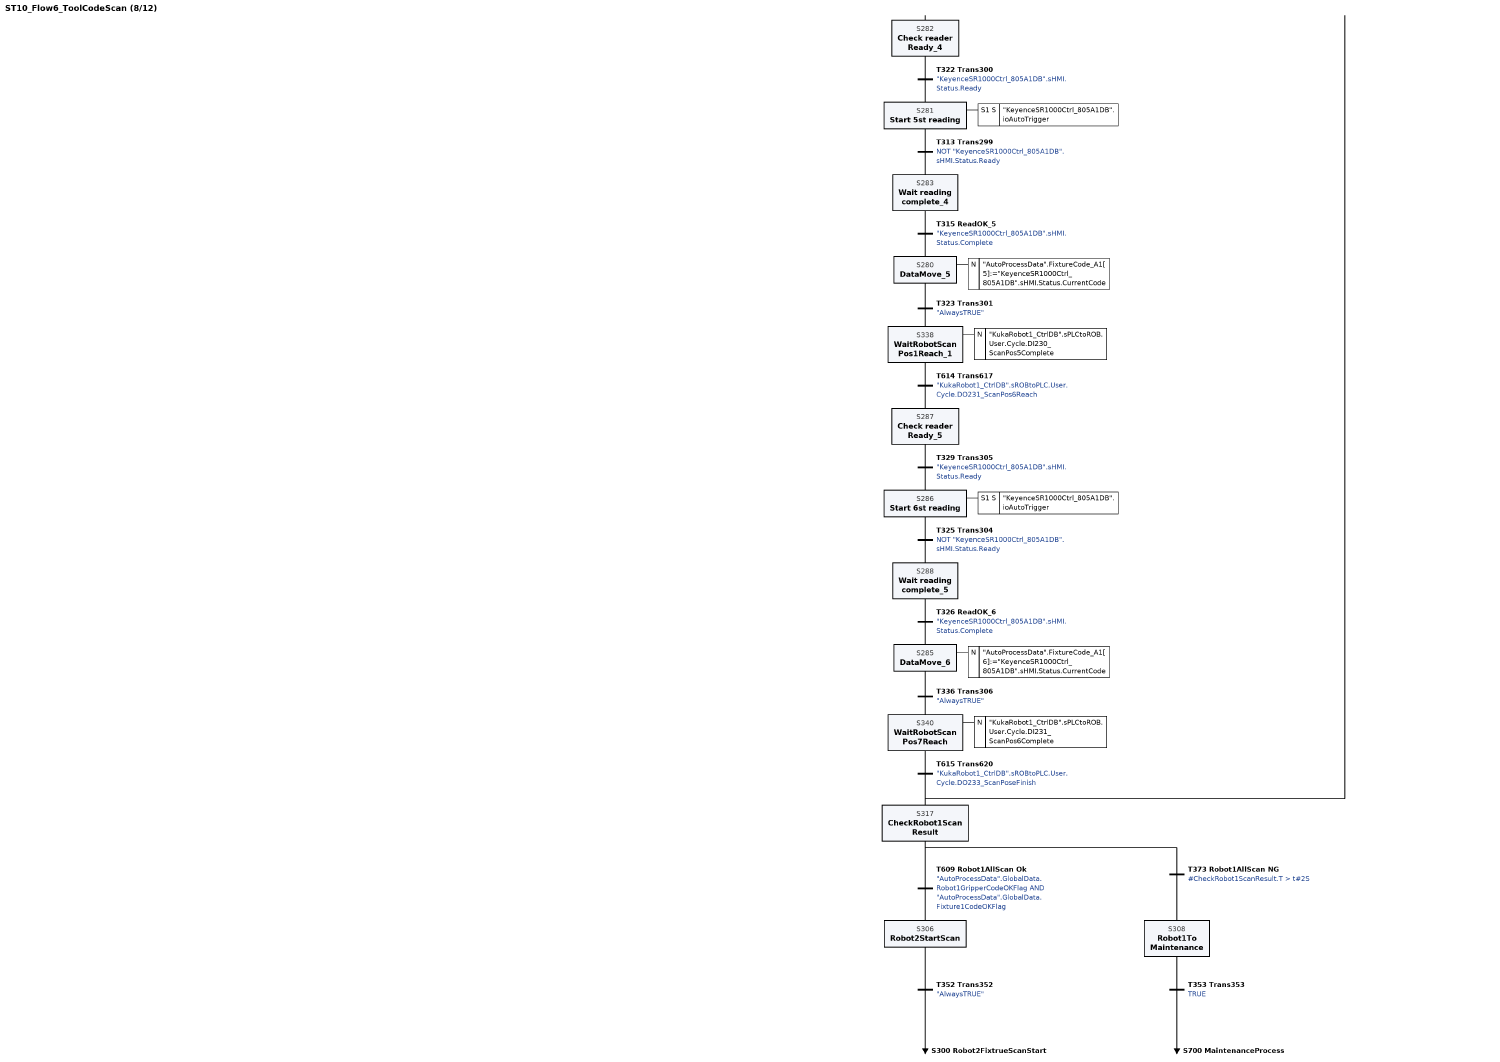
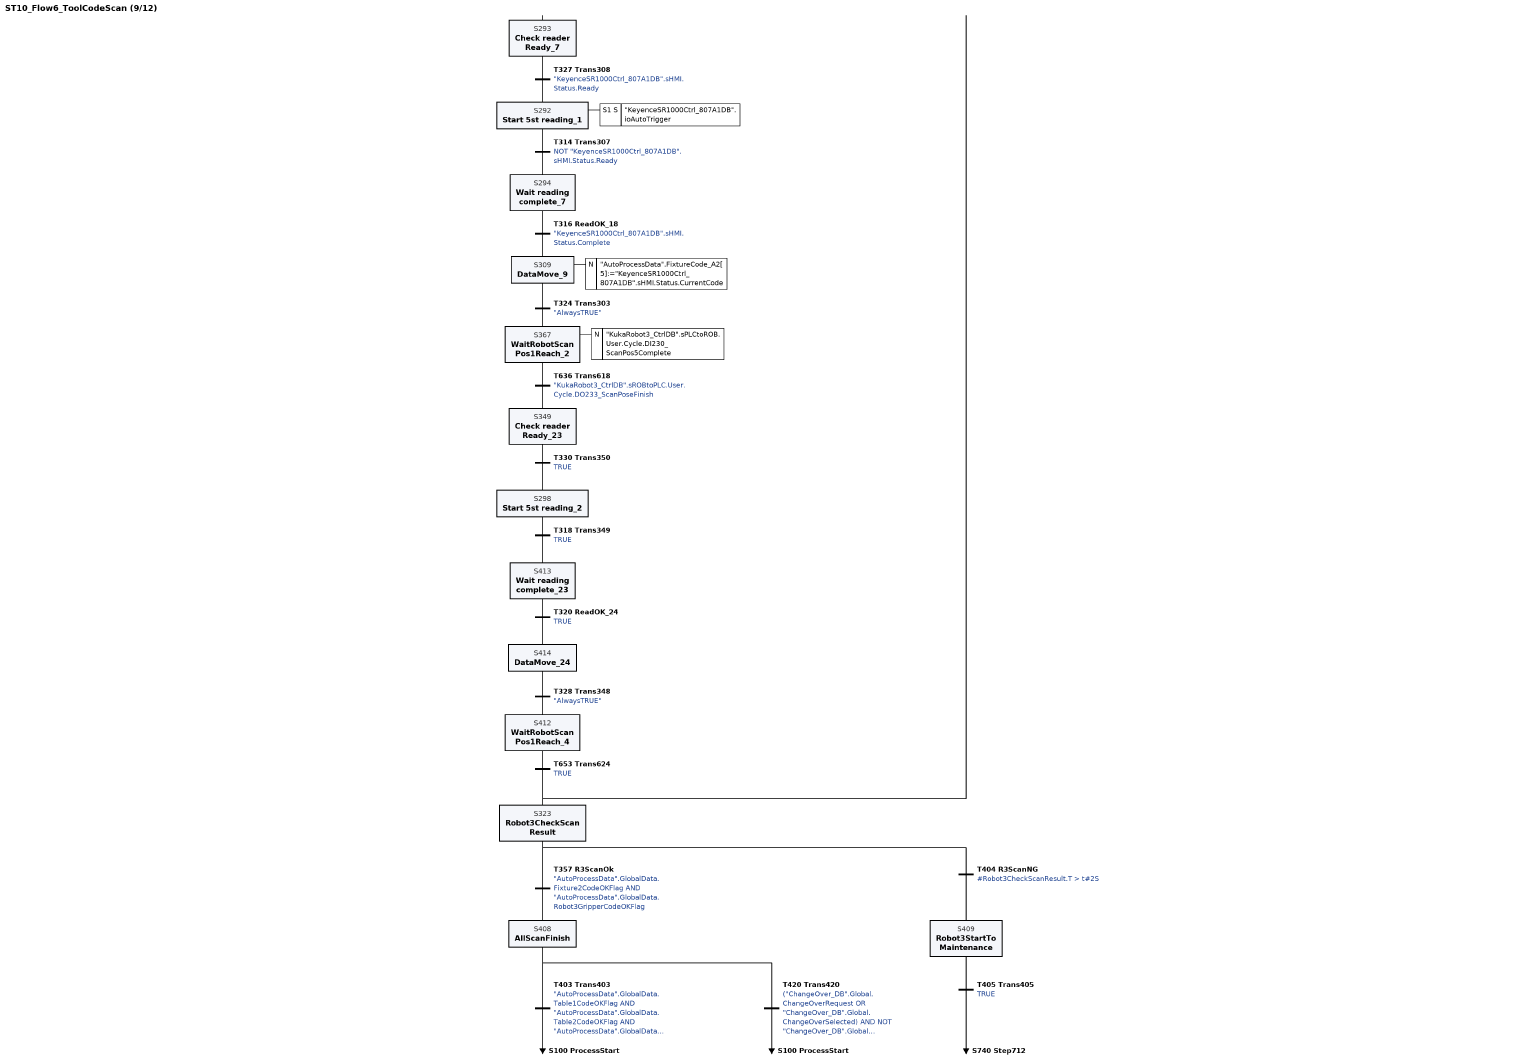
   // permanent pre-instructions
   NETWORK 1
      #TON[10].TON(IN := "AlwaysTRUE" AND "Station_Sys".Alarm.ImmediatelyStop, PT := T#300ms);
      #ioPM_Inface.AlarmImdilyStop := #TON[10].Q;
      #ioPM_Inface.AlarmCycleStop := "AlwaysTRUE" AND "Station_Sys".Alarm.CycleStop;
   NETWORK 2
      IF NOT False THEN
          #sCtrlMode(iSysInface := #iSysInface, ioPM_Inface := #ioPM_Inface, ioGraphCtrl := #RT_DATA.MOP);   // "SysFlowCtrlGraph"
      END_IF;
   NETWORK 3
      #TON[0].TON(IN := "AlwaysTRUE" AND "iA-Rotating product Check", PT := t#500ms);   // 工位11有托盘
      #TON[1].TOF(IN := "AlwaysTRUE" AND NOT "iA-Rotating product Check", PT := T#300ms);   // 工位无托盘
      #TON[2].TON(IN := "AlwaysTRUE", PT := T#300ms);
      #TON[3].TON(IN := "AlwaysTRUE", PT := T#300ms);
      #TON[4].TON(IN := "AlwaysTRUE", PT := T#300ms);
      #TON[5].TON(IN := "AlwaysTRUE", PT := T#300ms);
   NETWORK 4
      #前站站号 := 345;
      #本站站号 := 350;

   // sequencer 1: S01-S99 初始化 / S01-S99 Initial
   INITIAL_STEP F6_Initial:   // S1, max time T#10S, warning time T#7S
              S    #ioPM_Inface.InitialRun
              R    #ioPM_Inface.InitialOK
              R    #ioPM_Inface.WaitRunning
              R    #ioPM_Inface.Running
              R    #ioPM_Inface.UnPause
              R    "Station_Sys".Cmd.Calibration
              R    "Station_Sys".Cmd.ChangeOver
                   //"ST350_Sys".Cmd.DryRun
              R    "Station_Sys".Cmd.Reserve
              R    "Station_Sys".Cmd.OneCycle
              R    #ioPM_Inface.ProcessComplete
              R    #ioPM_Inface.ProcessStart
   END_STEP
   TRANSITION Trans1 FROM F6_Initial TO S2   // T1
      := #iSysInface.Ready;
   END_TRANSITION
   STEP S2:   // S2, max time T#10S, warning time T#7S
   END_STEP
   TRANSITION Trans2 FROM S2 TO S3   // T2
      := TRUE;
   END_TRANSITION
   STEP S4:   // S4, max time T#10S, warning time T#7S
   END_STEP
   TRANSITION Trans3 FROM S4 TO S5_MESInitial   // T3
      := TRUE;
   END_TRANSITION
   STEP S5_MESInitial:   // S5, max time T#10S, warning time T#7S
   END_STEP
   TRANSITION Trans325 FROM S5_MESInitial TO S8   // T4
      := TRUE;
   END_TRANSITION
   STEP S10_InitialFinish:   // S10, max time T#10S, warning time T#7S
              S    #ioPM_Inface.InitialOK
   END_STEP
   TRANSITION Trans102 FROM S10_InitialFinish TO ProcessStart   // T10, jump
      := #ioPM_Inface.Running;
   END_TRANSITION
   STEP S3:   // S3, max time T#10S, warning time T#7S
   END_STEP
   TRANSITION Trans613 FROM S3 TO S4   // T607
      := TRUE;
   END_TRANSITION
   STEP S8:   // S8, max time T#10S, warning time T#7S
   END_STEP
   TRANSITION Trans10 FROM S8 TO S9   // T8
      := TRUE;
   END_TRANSITION
   STEP S9:   // S9, max time T#10S, warning time T#7S
   END_STEP
   TRANSITION Trans7 FROM S9 TO S10_InitialFinish   // T9
      := TRUE;
   END_TRANSITION

   // sequencer 2: S100-S199 等待到位 / S100-S199 Fixture Scan Task
   STEP ProcessStart:   // S100, max time T#10S, warning time T#7S
      // 自动等待开始运行
              R    #ioPM_Inface.InitialRun
              R    #ioPM_Inface.ProcessComplete
              R    #ioPM_Inface.ProcessStart
              S    #ioPM_Inface.InitialOK
              S    #ioPM_Inface.WaitRunning
          S1  N    #ioPM_Inface.ProcessResult:=0
              R    "ST10_GeneralData".FlowControl_Handshake[6].Start
              R    "ST10_GeneralData".FlowControl_Handshake[6].Done
   END_STEP
   TRANSITION Trans200 FROM ProcessStart TO "WaitRobotBRAKETEST and MASTERINGTEST finish"   // T100
      := NOT #ioPM_Inface.AlarmCycleStop AND #ioPM_Inface.Running AND NOT #iSysInface.Auto.RunningOver AND (NOT #iSysInface.Auto.OneCycleMode OR (#iSysInface.Auto.OneCycleMode AND #ioPM_Inface.TriggerOneCycle));
   END_TRANSITION
   STEP "RB1_Process scan":   // S237, max time T#10S, warning time T#7S
              R    #ioPM_Inface.ProcessComplete
              S    #ioPM_Inface.ProcessStart
   END_STEP
   TRANSITION Trans250 FROM "RB1_Process scan" TO "Fixturecode reading"   // T249, jump
      := TRUE;
   END_TRANSITION
   STEP "Determine TableFixtureStatus":   // S101, max time T#10S, warning time T#7S
   END_STEP
   TRANSITION "Fixture NG" FROM "Determine TableFixtureStatus" TO WaitAllPartEmpty   // T101
      := ("ChangeOver_DB".Global.ScanFixtureFlag OR NOT "ChangeOver_DB".Global.AllFixtureScanCompareOk) AND NOT "ChangeOver_DB".Global.ChangeOverRequest AND NOT "ChangeOver_DB".Global.ChangeOverSelected;
   END_TRANSITION
   TRANSITION TaskMainten FROM "Determine TableFixtureStatus" TO RobotMaintenanceReq   // T110
      := "ChangeOver_DB".Global.ChangeOverRequest;
   END_TRANSITION
   STEP RobotMaintenanceReq:   // S102, max time T#10S, warning time T#7S
   END_STEP
   TRANSITION R1MaintenReady FROM RobotMaintenanceReq TO ClearAllBeltPallet   // T102
      := TRUE;
   END_TRANSITION
   STEP ToolScanCondition:   // S129, max time T#10S, warning time T#7S
   END_STEP
   TRANSITION Trans145 FROM ToolScanCondition TO "RB1_Process scan"   // T145
      := ("KukaRobot2_CtrlDB".sROBtoPLC.Sys.SO.IN_HOME OR "KukaRobot2_CtrlDB".sROBtoPLC.User.Cycle.DO298_MaintainFinish) AND NOT "KukaRobot2_CtrlDB".sROBtoPLC.User.Cycle.DO305_GripScanInside;
   END_TRANSITION
   STEP ClearAllBeltPallet:   // S417, max time T#10S, warning time T#7S
          S1  S    "AutoProcessControl".Global.ALL_EmptyPallet
          S0  R    "AutoProcessControl".Global.ALL_EmptyPallet
   END_STEP
   TRANSITION Trans414 FROM ClearAllBeltPallet TO MaintenanceProcess   // T414, jump
      := "ChangeOver_DB".Global.Station_empty AND "AutoProcessControl".Global.ALL_BeltPalletEmptyFinish;
   END_TRANSITION
   STEP WaitAllPartEmpty:   // S105, max time T#10S, warning time T#7S
   END_STEP
   TRANSITION "105ALL Empty" FROM WaitAllPartEmpty TO ToolScanCondition   // T105
      := "ChangeOver_DB".Global.Station_empty AND NOT "ChangeOver_DB".Global.ChangeOverRequest AND NOT "ChangeOver_DB".Global.ChangeOverSelected;
   END_TRANSITION
   TRANSITION Trans421 FROM WaitAllPartEmpty TO ProcessStart   // T421, jump
      := "ChangeOver_DB".Global.ChangeOverRequest OR "ChangeOver_DB".Global.ChangeOverSelected;
   END_TRANSITION
   STEP "WaitRobotBRAKETEST and MASTERINGTEST finish":   // S423, max time T#10S, warning time T#7S
   END_STEP
   TRANSITION Trans423 FROM "WaitRobotBRAKETEST and MASTERINGTEST finish" TO "Determine TableFixtureStatus"   // T423
      := NOT "KukaRobot1_CtrlDB".sROBtoPLC.User.Safety.DO452 AND NOT "KukaRobot1_CtrlDB".sROBtoPLC.User.Safety.DO460;
   END_TRANSITION

   // sequencer 3: S200-S299 Robot1 FixtureCode reading
   STEP "Fixturecode reading":   // S200, max time T#10S, warning time T#7S
              R    "KukaRobot1_CtrlDB".sPLCtoROB.User.Cycle.DI306_ScanPartComplete
              R    "KukaRobot1_CtrlDB".sPLCtoROB.User.Cycle.DI307_ScanPartFinish
              N    "AutoProcessData".GripperCode_R1[1]:=''
              N    "AutoProcessData".GripperCode_R1[2]:=''
              N    "AutoProcessData".GripperCode_R1[3]:=''
              N    "AutoProcessData".GripperCode_R1[4]:=''
              N    "AutoProcessData".FixtureCode_A1[1]:=''
              N    "AutoProcessData".FixtureCode_A1[2]:=''
              N    "AutoProcessData".FixtureCode_A1[3]:=''
              N    "AutoProcessData".FixtureCode_A1[4]:=''
              N    "AutoProcessData".FixtureCode_A1[5]:=''
              N    "AutoProcessData".FixtureCode_A1[6]:=''
              N    "AutoProcessData".FixtureCode_A1[7]:=''
              N    "AutoProcessData".FixtureCode_A1[8]:=''
   END_STEP
   TRANSITION Trans147 FROM "Fixturecode reading" TO CheckScanStatus   // T200
      := ("KukaRobot2_CtrlDB".sROBtoPLC.Sys.SO.IN_HOME OR "KukaRobot2_CtrlDB".sROBtoPLC.User.Cycle.DO298_MaintainFinish) AND NOT "KukaRobot2_CtrlDB".sROBtoPLC.User.Cycle.DO305_GripScanInside;
   END_TRANSITION
   STEP DataMove_2:   // S264, max time T#10S, warning time T#7S
              N    "AutoProcessData".FixtureCode_A1[2]:="KeyenceSR1000Ctrl_805A1DB".sHMI.Status.CurrentCode
   END_STEP
   TRANSITION Trans287 FROM DataMove_2 TO WaitRobotScanPos3Reach   // T290
      := "AlwaysTRUE";
   END_TRANSITION
   STEP Robot1ToMaintenance:   // S308, max time T#10S, warning time T#7S
   END_STEP
   TRANSITION Trans353 FROM Robot1ToMaintenance TO MaintenanceProcess   // T353, jump
      := TRUE;
   END_TRANSITION
   STEP CheckScanStatus:   // S208, max time T#10S, warning time T#7S
   END_STEP
   TRANSITION FixtureOk FROM CheckScanStatus TO WaitRobotScanStart   // T211
      := NOT "AutoProcessData".GlobalData.Robot1GripperCodeOKFlag;
   END_TRANSITION
   TRANSITION FixtureNG FROM CheckScanStatus TO Robot1FixtureScan   // T741
      := "AutoProcessData".GlobalData.Robot1GripperCodeOKFlag AND NOT "AutoProcessData".GlobalData.Fixture1CodeOKFlag;
   END_TRANSITION
   TRANSITION FixtureAllOk FROM CheckScanStatus TO CheckRobot1ScanResult   // T719
      := "AutoProcessData".GlobalData.Robot1GripperCodeOKFlag AND "AutoProcessData".GlobalData.Fixture1CodeOKFlag AND "KukaRobot2_CtrlDB".sROBtoPLC.Sys.SO.IN_HOME AND NOT "KukaRobot2_CtrlDB".sROBtoPLC.User.Cycle.DO305_GripScanInside;
   END_TRANSITION
   STEP DataMove_1:   // S263, max time T#10S, warning time T#7S
              N    "AutoProcessData".FixtureCode_A1[1]:="KeyenceSR1000Ctrl_805A1DB".sHMI.Status.CurrentCode
   END_STEP
   TRANSITION Trans283 FROM DataMove_1 TO WaitRobotScanPos2Reach   // T284
      := "AlwaysTRUE";
   END_TRANSITION
   STEP WaitRobotScanStart:   // S311, max time T#10S, warning time T#7S
              N    "AutoProcessControl".Robot_1.GripScanRequest
   END_STEP
   TRANSITION Trans606 FROM WaitRobotScanStart TO WaitRobotScanGripPos1Reach   // T606
      := NOT "KukaRobot1_CtrlDB".sROBtoPLC.User.Cycle.DO225_ScanPosInside AND "KukaRobot1_CtrlDB".sROBtoPLC.User.Cycle.DO305_GripScanInside;
   END_TRANSITION
   STEP "Start 1st reading":   // S265, max time T#10S, warning time T#7S
          S1  S    "KeyenceSR1000Ctrl_805A1DB".ioAutoTrigger
   END_STEP
   TRANSITION Trans282 FROM "Start 1st reading" TO "Wait reading complete"   // T282
      := NOT "KeyenceSR1000Ctrl_805A1DB".sHMI.Status.Ready;
   END_TRANSITION
   STEP "Check reader Ready":   // S266, max time T#10S, warning time T#7S
   END_STEP
   TRANSITION Trans279 FROM "Check reader Ready" TO "Start 1st reading"   // T281
      := "KeyenceSR1000Ctrl_805A1DB".sHMI.Status.Ready;
   END_TRANSITION
   STEP "Wait reading complete":   // S267, max time T#10S, warning time T#7S
   END_STEP
   TRANSITION ReadOK_1 FROM "Wait reading complete" TO DataMove_1   // T280
      := "KeyenceSR1000Ctrl_805A1DB".sHMI.Status.Complete;
   END_TRANSITION
   STEP "Wait reading complete_5":   // S288, max time T#10S, warning time T#7S
   END_STEP
   TRANSITION ReadOK_6 FROM "Wait reading complete_5" TO DataMove_6   // T326
      := "KeyenceSR1000Ctrl_805A1DB".sHMI.Status.Complete;
   END_TRANSITION
   STEP "Check reader Ready_5":   // S287, max time T#10S, warning time T#7S
   END_STEP
   TRANSITION Trans305 FROM "Check reader Ready_5" TO "Start 6st reading"   // T329
      := "KeyenceSR1000Ctrl_805A1DB".sHMI.Status.Ready;
   END_TRANSITION
   STEP "Start 6st reading":   // S286, max time T#10S, warning time T#7S
          S1  S    "KeyenceSR1000Ctrl_805A1DB".ioAutoTrigger
   END_STEP
   TRANSITION Trans304 FROM "Start 6st reading" TO "Wait reading complete_5"   // T325
      := NOT "KeyenceSR1000Ctrl_805A1DB".sHMI.Status.Ready;
   END_TRANSITION
   STEP WaitRobotScanPos1Reach_1:   // S338, max time T#10S, warning time T#7S
              N    "KukaRobot1_CtrlDB".sPLCtoROB.User.Cycle.DI230_ScanPos5Complete
   END_STEP
   TRANSITION Trans617 FROM WaitRobotScanPos1Reach_1 TO "Check reader Ready_5"   // T614
      := "KukaRobot1_CtrlDB".sROBtoPLC.User.Cycle.DO231_ScanPos6Reach;
   END_TRANSITION
   STEP WaitRobotScanPos5Reach:   // S336, max time T#10S, warning time T#7S
              N    "KukaRobot1_CtrlDB".sPLCtoROB.User.Cycle.DI229_ScanPos4Complete
   END_STEP
   TRANSITION Trans616 FROM WaitRobotScanPos5Reach TO WaitServoStop   // T613
      := "KukaRobot1_CtrlDB".sROBtoPLC.User.Cycle.DO230_ScanPos5Reach;
   END_TRANSITION
   STEP DataMove_6:   // S285, max time T#10S, warning time T#7S
              N    "AutoProcessData".FixtureCode_A1[6]:="KeyenceSR1000Ctrl_805A1DB".sHMI.Status.CurrentCode
   END_STEP
   TRANSITION Trans306 FROM DataMove_6 TO WaitRobotScanPos7Reach   // T336
      := "AlwaysTRUE";
   END_TRANSITION
   STEP WaitRobotScanPos2Reach:   // S330, max time T#10S, warning time T#7S
              N    "KukaRobot1_CtrlDB".sPLCtoROB.User.Cycle.DI226_ScanPos1Complete
   END_STEP
   TRANSITION Trans612 FROM WaitRobotScanPos2Reach TO "Check reader Ready_1"   // T610
      := "KukaRobot1_CtrlDB".sROBtoPLC.User.Cycle.DO227_ScanPos2Reach;
   END_TRANSITION
   STEP WaitRobotScanPos4Reach:   // S334, max time T#10S, warning time T#7S
              N    "KukaRobot1_CtrlDB".sPLCtoROB.User.Cycle.DI228_ScanPos3Complete
   END_STEP
   TRANSITION Trans615 FROM WaitRobotScanPos4Reach TO "Check reader Ready_3"   // T612
      := "KukaRobot1_CtrlDB".sROBtoPLC.User.Cycle.DO229_ScanPos4Reach;
   END_TRANSITION
   STEP "Start 5st reading":   // S281, max time T#10S, warning time T#7S
          S1  S    "KeyenceSR1000Ctrl_805A1DB".ioAutoTrigger
   END_STEP
   TRANSITION Trans299 FROM "Start 5st reading" TO "Wait reading complete_4"   // T313
      := NOT "KeyenceSR1000Ctrl_805A1DB".sHMI.Status.Ready;
   END_TRANSITION
   STEP "Check reader Ready_4":   // S282, max time T#10S, warning time T#7S
   END_STEP
   TRANSITION Trans300 FROM "Check reader Ready_4" TO "Start 5st reading"   // T322
      := "KeyenceSR1000Ctrl_805A1DB".sHMI.Status.Ready;
   END_TRANSITION
   STEP "Wait reading complete_4":   // S283, max time T#10S, warning time T#7S
   END_STEP
   TRANSITION ReadOK_5 FROM "Wait reading complete_4" TO DataMove_5   // T315
      := "KeyenceSR1000Ctrl_805A1DB".sHMI.Status.Complete;
   END_TRANSITION
   STEP "Wait reading complete_3":   // S278, max time T#10S, warning time T#7S
   END_STEP
   TRANSITION ReadOK_4 FROM "Wait reading complete_3" TO DataMove_4   // T299
      := "KeyenceSR1000Ctrl_805A1DB".sHMI.Status.Complete;
   END_TRANSITION
   STEP "Check reader Ready_3":   // S277, max time T#10S, warning time T#7S
   END_STEP
   TRANSITION Trans296 FROM "Check reader Ready_3" TO "Start 4st reading"   // T306
      := "KeyenceSR1000Ctrl_805A1DB".sHMI.Status.Ready;
   END_TRANSITION
   STEP DataMove_5:   // S280, max time T#10S, warning time T#7S
              N    "AutoProcessData".FixtureCode_A1[5]:="KeyenceSR1000Ctrl_805A1DB".sHMI.Status.CurrentCode
   END_STEP
   TRANSITION Trans301 FROM DataMove_5 TO WaitRobotScanPos1Reach_1   // T323
      := "AlwaysTRUE";
   END_TRANSITION
   STEP DataMove_4:   // S275, max time T#10S, warning time T#7S
              N    "AutoProcessData".FixtureCode_A1[4]:="KeyenceSR1000Ctrl_805A1DB".sHMI.Status.CurrentCode
   END_STEP
   TRANSITION Trans297 FROM DataMove_4 TO WaitRobotScanPos5Reach   // T307
      := "AlwaysTRUE";
   END_TRANSITION
   STEP "Start 4st reading":   // S276, max time T#10S, warning time T#7S
          S1  S    "KeyenceSR1000Ctrl_805A1DB".ioAutoTrigger
   END_STEP
   TRANSITION Trans295 FROM "Start 4st reading" TO "Wait reading complete_3"   // T298
      := NOT "KeyenceSR1000Ctrl_805A1DB".sHMI.Status.Ready;
   END_TRANSITION
   STEP "Check reader Ready_2":   // S273, max time T#10S, warning time T#7S
   END_STEP
   TRANSITION Trans292 FROM "Check reader Ready_2" TO "Start 3st reading"   // T295
      := "KeyenceSR1000Ctrl_805A1DB".sHMI.Status.Ready;
   END_TRANSITION
   STEP "Wait reading complete_2":   // S274, max time T#10S, warning time T#7S
   END_STEP
   TRANSITION ReadOK_3 FROM "Wait reading complete_2" TO DataMove_3   // T293
      := "KeyenceSR1000Ctrl_805A1DB".sHMI.Status.Complete;
   END_TRANSITION
   STEP WaitRobotScanPos3Reach:   // S332, max time T#10S, warning time T#7S
              N    "KukaRobot1_CtrlDB".sPLCtoROB.User.Cycle.DI227_ScanPos2Complete
   END_STEP
   TRANSITION Trans614 FROM WaitRobotScanPos3Reach TO "Check reader Ready_2"   // T611
      := "KukaRobot1_CtrlDB".sROBtoPLC.User.Cycle.DO228_ScanPos3Reach;
   END_TRANSITION
   STEP "Check reader Ready_1":   // S269, max time T#10S, warning time T#7S
   END_STEP
   TRANSITION Trans286 FROM "Check reader Ready_1" TO "Start 2st reading"   // T289
      := "KeyenceSR1000Ctrl_805A1DB".sHMI.Status.Ready;
   END_TRANSITION
   STEP "Wait reading complete_1":   // S270, max time T#10S, warning time T#7S
   END_STEP
   TRANSITION ReadOK_2 FROM "Wait reading complete_1" TO DataMove_2   // T287
      := "KeyenceSR1000Ctrl_805A1DB".sHMI.Status.Complete;
   END_TRANSITION
   STEP DataMove_3:   // S271, max time T#10S, warning time T#7S
              N    "AutoProcessData".FixtureCode_A1[3]:="KeyenceSR1000Ctrl_805A1DB".sHMI.Status.CurrentCode
   END_STEP
   TRANSITION Trans293 FROM DataMove_3 TO WaitRobotScanPos4Reach   // T296
      := "AlwaysTRUE";
   END_TRANSITION
   STEP "Start 3st reading":   // S272, max time T#10S, warning time T#7S
          S1  S    "KeyenceSR1000Ctrl_805A1DB".ioAutoTrigger
   END_STEP
   TRANSITION Trans291 FROM "Start 3st reading" TO "Wait reading complete_2"   // T292
      := NOT "KeyenceSR1000Ctrl_805A1DB".sHMI.Status.Ready;
   END_TRANSITION
   STEP "Start 2st reading":   // S268, max time T#10S, warning time T#7S
          S1  S    "KeyenceSR1000Ctrl_805A1DB".ioAutoTrigger
   END_STEP
   TRANSITION Trans285 FROM "Start 2st reading" TO "Wait reading complete_1"   // T286
      := NOT "KeyenceSR1000Ctrl_805A1DB".sHMI.Status.Ready;
   END_TRANSITION
   STEP Robot2StartScan:   // S306, max time T#10S, warning time T#7S
   END_STEP
   TRANSITION Trans352 FROM Robot2StartScan TO Robot2FixtrueScanStart   // T352, jump
      := "AlwaysTRUE";
   END_TRANSITION
   STEP WaitRobotScanPos1Reach:   // S316, max time T#10S, warning time T#7S
   END_STEP
   TRANSITION Trans608 FROM WaitRobotScanPos1Reach TO "Check reader Ready"   // T608
      := "KukaRobot1_CtrlDB".sROBtoPLC.User.Cycle.DO226_ScanPos1Reach;
   END_TRANSITION
   STEP WaitRobotScanPos7Reach:   // S340, max time T#10S, warning time T#7S
              N    "KukaRobot1_CtrlDB".sPLCtoROB.User.Cycle.DI231_ScanPos6Complete
   END_STEP
   TRANSITION Trans620 FROM WaitRobotScanPos7Reach TO CheckRobot1ScanResult   // T615
      := "KukaRobot1_CtrlDB".sROBtoPLC.User.Cycle.DO233_ScanPoseFinish;
   END_TRANSITION
   STEP CheckRobot1ScanResult:   // S317, max time T#10S, warning time T#7S
   END_STEP
   TRANSITION "Robot1AllScan Ok" FROM CheckRobot1ScanResult TO Robot2StartScan   // T609
      := "AutoProcessData".GlobalData.Robot1GripperCodeOKFlag AND "AutoProcessData".GlobalData.Fixture1CodeOKFlag;
   END_TRANSITION
   TRANSITION "Robot1AllScan NG" FROM CheckRobot1ScanResult TO Robot1ToMaintenance   // T373
      := #CheckRobot1ScanResult.T > t#2S;
   END_TRANSITION
   STEP WaitRobotScanGripPos1Reach:   // S329, max time T#10S, warning time T#7S
   END_STEP
   TRANSITION Trans607 FROM WaitRobotScanGripPos1Reach TO "Check reader Ready_10"   // T617
      := "KukaRobot1_CtrlDB".sROBtoPLC.User.Cycle.DO307_ScanPos1Reach;
   END_TRANSITION
   STEP "Check reader Ready_10":   // S331, max time T#10S, warning time T#7S
   END_STEP
   TRANSITION Trans629 FROM "Check reader Ready_10" TO "Start 10st reading"   // T618
      := "KeyenceSR1000Ctrl_804A1DB".oReady;
   END_TRANSITION
   STEP "Start 10st reading":   // S333, max time T#10S, warning time T#7S
          S1  S    "KeyenceSR1000Ctrl_804A1DB".ioAutoTrigger
   END_STEP
   TRANSITION Trans630 FROM "Start 10st reading" TO "Wait reading complete_10"   // T619
      := NOT "KeyenceSR1000Ctrl_804A1DB".sHMI.Status.Ready;
   END_TRANSITION
   STEP Robot1FixtureScan:   // S335, max time T#10S, warning time T#7S
              N    "AutoProcessControl".Fixture1Code.Robot1CodeReadReq
   END_STEP
   TRANSITION Trans631 FROM Robot1FixtureScan TO WaitRobotScanPos1Reach   // T620
      := "KukaRobot1_CtrlDB".sROBtoPLC.User.Cycle.DO225_ScanPosInside AND NOT "KukaRobot1_CtrlDB".sROBtoPLC.User.Cycle.DO305_GripScanInside;
   END_TRANSITION
   STEP "Wait reading complete_10":   // S295, max time T#10S, warning time T#7S
   END_STEP
   TRANSITION ReadOK_10 FROM "Wait reading complete_10" TO DataMove_10   // T351
      := "KeyenceSR1000Ctrl_804A1DB".sHMI.Status.Complete;
   END_TRANSITION
   STEP DataMove_10:   // S296, max time T#10S, warning time T#7S
              N    "AutoProcessData".GripperCode_R1[1]:="KeyenceSR1000Ctrl_804A1DB".sHMI.Status.CurrentCode
   END_STEP
   TRANSITION Trans313 FROM DataMove_10 TO RobotScanGripPos1Comp   // T355
      := TRUE;
   END_TRANSITION
   STEP RobotScanGripPos1Comp:   // S299, max time T#10S, warning time T#7S
              R    "KukaRobot1_CtrlDB".sPLCtoROB.User.Cycle.DI307_ScanPartFinish
              N    "KukaRobot1_CtrlDB".sPLCtoROB.User.Cycle.DI306_ScanPartComplete
   END_STEP
   TRANSITION Trans314 FROM RobotScanGripPos1Comp TO WaitRobotScanGripPos2Reach   // T359
      := NOT "KukaRobot1_CtrlDB".sROBtoPLC.User.Cycle.DO307_ScanPos1Reach;
   END_TRANSITION
   STEP WaitRobotScanGripPos2Reach:   // S304, max time T#10S, warning time T#7S
   END_STEP
   TRANSITION Trans316 FROM WaitRobotScanGripPos2Reach TO "Check reader Ready_11"   // T360
      := "KukaRobot1_CtrlDB".sROBtoPLC.User.Cycle.DO308_ScanPos2Reach;
   END_TRANSITION
   STEP "Check reader Ready_11":   // S337, max time T#10S, warning time T#7S
   END_STEP
   TRANSITION Trans632 FROM "Check reader Ready_11" TO "Start 11st reading"   // T621
      := "KeyenceSR1000Ctrl_804A1DB".oReady;
   END_TRANSITION
   STEP "Start 11st reading":   // S339, max time T#10S, warning time T#7S
          S1  S    "KeyenceSR1000Ctrl_804A1DB".ioAutoTrigger
   END_STEP
   TRANSITION Trans633 FROM "Start 11st reading" TO "Wait reading complete_11"   // T622
      := NOT "KeyenceSR1000Ctrl_804A1DB".sHMI.Status.Ready;
   END_TRANSITION
   STEP "Wait reading complete_11":   // S342, max time T#10S, warning time T#7S
   END_STEP
   TRANSITION ReadOK_11 FROM "Wait reading complete_11" TO DataMove_11   // T361
      := "KeyenceSR1000Ctrl_804A1DB".sHMI.Status.Complete;
   END_TRANSITION
   STEP DataMove_11:   // S343, max time T#10S, warning time T#7S
              N    "AutoProcessData".GripperCode_R1[2]:="KeyenceSR1000Ctrl_804A1DB".sHMI.Status.CurrentCode
   END_STEP
   TRANSITION Trans318 FROM DataMove_11 TO RobotScanGripPos2Comp   // T364
      := TRUE;
   END_TRANSITION
   STEP RobotScanGripPos2Comp:   // S345, max time T#10S, warning time T#7S
              R    "KukaRobot1_CtrlDB".sPLCtoROB.User.Cycle.DI307_ScanPartFinish
              N    "KukaRobot1_CtrlDB".sPLCtoROB.User.Cycle.DI306_ScanPartComplete
   END_STEP
   TRANSITION Trans319 FROM RobotScanGripPos2Comp TO WaitRobotScanGripPos3Reach   // T367
      := NOT "KukaRobot1_CtrlDB".sROBtoPLC.User.Cycle.DO308_ScanPos2Reach;
   END_TRANSITION
   STEP WaitRobotScanGripPos3Reach:   // S346, max time T#10S, warning time T#7S
   END_STEP
   TRANSITION Trans320 FROM WaitRobotScanGripPos3Reach TO "Check reader Ready_12"   // T368
      := "KukaRobot1_CtrlDB".sROBtoPLC.User.Cycle.DO309_ScanPos3Reach;
   END_TRANSITION
   STEP "Check reader Ready_12":   // S347, max time T#10S, warning time T#7S
   END_STEP
   TRANSITION Trans634 FROM "Check reader Ready_12" TO "Start 11st reading_1"   // T623
      := "KeyenceSR1000Ctrl_804A1DB".oReady;
   END_TRANSITION
   STEP "Start 11st reading_1":   // S348, max time T#10S, warning time T#7S
          S1  S    "KeyenceSR1000Ctrl_804A1DB".ioAutoTrigger
   END_STEP
   TRANSITION Trans635 FROM "Start 11st reading_1" TO "Wait reading complete_12"   // T624
      := NOT "KeyenceSR1000Ctrl_804A1DB".sHMI.Status.Ready;
   END_TRANSITION
   STEP "Wait reading complete_12":   // S350, max time T#10S, warning time T#7S
   END_STEP
   TRANSITION ReadOK_12 FROM "Wait reading complete_12" TO DataMove_12   // T369
      := "KeyenceSR1000Ctrl_804A1DB".sHMI.Status.Complete;
   END_TRANSITION
   STEP DataMove_12:   // S351, max time T#10S, warning time T#7S
              N    "AutoProcessData".GripperCode_R1[3]:="KeyenceSR1000Ctrl_804A1DB".sHMI.Status.CurrentCode
   END_STEP
   TRANSITION Trans322 FROM DataMove_12 TO RobotScanGripPos3Comp   // T372
      := TRUE;
   END_TRANSITION
   STEP RobotScanGripPos3Comp:   // S353, max time T#10S, warning time T#7S
              R    "KukaRobot1_CtrlDB".sPLCtoROB.User.Cycle.DI307_ScanPartFinish
              N    "KukaRobot1_CtrlDB".sPLCtoROB.User.Cycle.DI306_ScanPartComplete
   END_STEP
   TRANSITION Trans323 FROM RobotScanGripPos3Comp TO WaitRobotScanGripPos4Reach   // T375
      := NOT "KukaRobot1_CtrlDB".sROBtoPLC.User.Cycle.DO309_ScanPos3Reach;
   END_TRANSITION
   STEP WaitRobotScanGripPos4Reach:   // S354, max time T#10S, warning time T#7S
   END_STEP
   TRANSITION Trans324 FROM WaitRobotScanGripPos4Reach TO "Check reader Ready_13"   // T376
      := "KukaRobot1_CtrlDB".sROBtoPLC.User.Cycle.DO310_ScanPos4Reach;
   END_TRANSITION
   STEP "Check reader Ready_13":   // S355, max time T#10S, warning time T#7S
   END_STEP
   TRANSITION Trans636 FROM "Check reader Ready_13" TO "Start 11st reading_2"   // T625
      := "KeyenceSR1000Ctrl_804A1DB".oReady;
   END_TRANSITION
   STEP "Start 11st reading_2":   // S356, max time T#10S, warning time T#7S
          S1  S    "KeyenceSR1000Ctrl_804A1DB".ioAutoTrigger
   END_STEP
   TRANSITION Trans637 FROM "Start 11st reading_2" TO "Wait reading complete_13"   // T626
      := NOT "KeyenceSR1000Ctrl_804A1DB".sHMI.Status.Ready;
   END_TRANSITION
   STEP "Wait reading complete_13":   // S358, max time T#10S, warning time T#7S
   END_STEP
   TRANSITION ReadOK_13 FROM "Wait reading complete_13" TO DataMove_13   // T377
      := "KeyenceSR1000Ctrl_804A1DB".sHMI.Status.Complete;
   END_TRANSITION
   STEP DataMove_13:   // S359, max time T#10S, warning time T#7S
              N    "AutoProcessData".GripperCode_R1[4]:="KeyenceSR1000Ctrl_804A1DB".sHMI.Status.CurrentCode
   END_STEP
   TRANSITION Trans327 FROM DataMove_13 TO RobotScanGripPos4Comp   // T380
      := TRUE;
   END_TRANSITION
   STEP RobotScanGripPos4Comp:   // S361, max time T#10S, warning time T#7S
              N    "KukaRobot1_CtrlDB".sPLCtoROB.User.Cycle.DI307_ScanPartFinish
              N    "KukaRobot1_CtrlDB".sPLCtoROB.User.Cycle.DI306_ScanPartComplete
   END_STEP
   TRANSITION Trans328 FROM RobotScanGripPos4Comp TO Robot1FixtureScan   // T383
      := "KukaRobot1_CtrlDB".sROBtoPLC.User.Cycle.DO306_GripScanFinish;
   END_TRANSITION
   STEP WaitServoStop:   // S422, max time T#10S, warning time T#7S
   END_STEP
   TRANSITION Trans422 FROM WaitServoStop TO "Check reader Ready_4"   // T422
      := "iC-GlueServoHomePos";
   END_TRANSITION

   // sequencer 4: S600-S699工件放行 / S300-S399 Robot2 FixtureCode reading
   STEP Robot2FixtrueScanStart:   // S300, max time T#10S, warning time T#7S
              R    "KukaRobot2_CtrlDB".sPLCtoROB.User.Cycle.DI307_ScanPartFinish
              R    "KukaRobot2_CtrlDB".sPLCtoROB.User.Cycle.DI306_ScanPartComplete
              N    "AutoProcessData".GripperCode_R2[1]:=''
              N    "AutoProcessData".GripperCode_R2[2]:=''
              N    "AutoProcessData".GripperCode_R2[3]:=''
              N    "AutoProcessData".GripperCode_R2[4]:=''
   END_STEP
   TRANSITION Trans302 FROM Robot2FixtrueScanStart TO Robot2CheckScanStatus   // T300
      := ("KukaRobot1_CtrlDB".sROBtoPLC.Sys.SO.IN_HOME OR "KukaRobot1_CtrlDB".sROBtoPLC.User.Cycle.DO298_MaintainFinish) AND (NOT "KukaRobot1_CtrlDB".sROBtoPLC.User.Cycle.DO225_ScanPosInside OR "KukaRobot1_CtrlDB".sROBtoPLC.Sys.SO.IN_HOME);
   END_TRANSITION
   STEP "Check reader Ready_14":   // S341, max time T#10S, warning time T#7S
   END_STEP
   TRANSITION Trans638 FROM "Check reader Ready_14" TO "Start 10st reading_1"   // T627
      := "KeyenceSR1000Ctrl_806A1DB".oReady;
   END_TRANSITION
   STEP Robot2CheckScanResult:   // S149, max time T#10S, warning time T#7S
   END_STEP
   TRANSITION R2ScanOk FROM Robot2CheckScanResult TO Robot3StartToScan   // T149
      := "AutoProcessData".GlobalData.Robot2GripperCodeOKFlag;
   END_TRANSITION
   TRANSITION R2ScanNG FROM Robot2CheckScanResult TO Robot2StartToMaintenanc   // T675
      := NOT "AutoProcessData".GlobalData.Robot2GripperCodeOKFlag AND (#Robot2CheckScanResult.T > t#2S);
   END_TRANSITION
   STEP Robot3StartToScan:   // S365, max time T#10S, warning time T#7S
   END_STEP
   TRANSITION Trans674 FROM Robot3StartToScan TO Robot3FixtrueScanStart   // T674, jump
      := NOT "KukaRobot2_CtrlDB".sROBtoPLC.User.Cycle.DO297_MaintainInside;
   END_TRANSITION
   STEP Robot2StartToMaintenanc:   // S366, max time T#10S, warning time T#7S
   END_STEP
   TRANSITION Trans678 FROM Robot2StartToMaintenanc TO Step720   // T676, jump
      := TRUE;
   END_TRANSITION
   STEP "Start 10st reading_1":   // S344, max time T#10S, warning time T#7S
          S1  S    "KeyenceSR1000Ctrl_806A1DB".ioAutoTrigger
   END_STEP
   TRANSITION Trans642 FROM "Start 10st reading_1" TO "Wait reading complete_14"   // T628
      := NOT "KeyenceSR1000Ctrl_806A1DB".sHMI.Status.Ready;
   END_TRANSITION
   STEP "Wait reading complete_14":   // S297, max time T#10S, warning time T#7S
   END_STEP
   TRANSITION ReadOK_14 FROM "Wait reading complete_14" TO DataMove_14   // T354
      := "KeyenceSR1000Ctrl_806A1DB".sHMI.Status.Complete;
   END_TRANSITION
   STEP DataMove_14:   // S303, max time T#10S, warning time T#7S
              N    "AutoProcessData".GripperCode_R2[1]:="KeyenceSR1000Ctrl_806A1DB".sHMI.Status.CurrentCode
   END_STEP
   TRANSITION Trans315 FROM DataMove_14 TO RobotScanGripPos1Comp_1   // T356
      := "AlwaysTRUE";
   END_TRANSITION
   STEP RobotScanGripPos1Comp_1:   // S305, max time T#10S, warning time T#7S
              R    "KukaRobot2_CtrlDB".sPLCtoROB.User.Cycle.DI307_ScanPartFinish
              N    "KukaRobot2_CtrlDB".sPLCtoROB.User.Cycle.DI306_ScanPartComplete
   END_STEP
   TRANSITION Trans317 FROM RobotScanGripPos1Comp_1 TO WaitRobotScanGripPos2Reach_1   // T362
      := NOT "KukaRobot2_CtrlDB".sROBtoPLC.User.Cycle.DO307_ScanPos1Reach;
   END_TRANSITION
   STEP WaitRobotScanGripPos2Reach_1:   // S307, max time T#10S, warning time T#7S
   END_STEP
   TRANSITION Trans321 FROM WaitRobotScanGripPos2Reach_1 TO "Check reader Ready_15"   // T363
      := "KukaRobot2_CtrlDB".sROBtoPLC.User.Cycle.DO308_ScanPos2Reach;
   END_TRANSITION
   STEP "Check reader Ready_15":   // S352, max time T#10S, warning time T#7S
   END_STEP
   TRANSITION Trans652 FROM "Check reader Ready_15" TO "Start 11st reading_3"   // T630
      := "KeyenceSR1000Ctrl_806A1DB".oReady;
   END_TRANSITION
   STEP "Start 11st reading_3":   // S357, max time T#10S, warning time T#7S
          S1  S    "KeyenceSR1000Ctrl_806A1DB".ioAutoTrigger
   END_STEP
   TRANSITION Trans653 FROM "Start 11st reading_3" TO "Wait reading complete_15"   // T631
      := NOT "KeyenceSR1000Ctrl_806A1DB".sHMI.Status.Ready;
   END_TRANSITION
   STEP "Wait reading complete_15":   // S360, max time T#10S, warning time T#7S
   END_STEP
   TRANSITION ReadOK_15 FROM "Wait reading complete_15" TO DataMove_15   // T365
      := "KeyenceSR1000Ctrl_806A1DB".sHMI.Status.Complete;
   END_TRANSITION
   STEP DataMove_15:   // S362, max time T#10S, warning time T#7S
              N    "AutoProcessData".GripperCode_R2[2]:="KeyenceSR1000Ctrl_806A1DB".sHMI.Status.CurrentCode
   END_STEP
   TRANSITION Trans326 FROM DataMove_15 TO RobotScanGripPos2Comp_1   // T366
      := "AlwaysTRUE";
   END_TRANSITION
   STEP RobotScanGripPos2Comp_1:   // S371, max time T#10S, warning time T#7S
              R    "KukaRobot2_CtrlDB".sPLCtoROB.User.Cycle.DI307_ScanPartFinish
              N    "KukaRobot2_CtrlDB".sPLCtoROB.User.Cycle.DI306_ScanPartComplete
   END_STEP
   TRANSITION Trans329 FROM RobotScanGripPos2Comp_1 TO WaitRobotScanGripPos3Reach_1   // T370
      := NOT "KukaRobot2_CtrlDB".sROBtoPLC.User.Cycle.DO308_ScanPos2Reach;
   END_TRANSITION
   STEP WaitRobotScanGripPos3Reach_1:   // S372, max time T#10S, warning time T#7S
   END_STEP
   TRANSITION Trans330 FROM WaitRobotScanGripPos3Reach_1 TO "Check reader Ready_16"   // T371
      := "KukaRobot2_CtrlDB".sROBtoPLC.User.Cycle.DO309_ScanPos3Reach;
   END_TRANSITION
   STEP "Check reader Ready_16":   // S373, max time T#10S, warning time T#7S
   END_STEP
   TRANSITION Trans673 FROM "Check reader Ready_16" TO "Start 11st reading_4"   // T632
      := "KeyenceSR1000Ctrl_806A1DB".oReady;
   END_TRANSITION
   STEP "Start 11st reading_4":   // S374, max time T#10S, warning time T#7S
          S1  S    "KeyenceSR1000Ctrl_806A1DB".ioAutoTrigger
   END_STEP
   TRANSITION Trans675 FROM "Start 11st reading_4" TO "Wait reading complete_16"   // T633
      := NOT "KeyenceSR1000Ctrl_806A1DB".sHMI.Status.Ready;
   END_TRANSITION
   STEP "Wait reading complete_16":   // S375, max time T#10S, warning time T#7S
   END_STEP
   TRANSITION ReadOK_16 FROM "Wait reading complete_16" TO DataMove_16   // T374
      := "KeyenceSR1000Ctrl_806A1DB".sHMI.Status.Complete;
   END_TRANSITION
   STEP DataMove_16:   // S376, max time T#10S, warning time T#7S
              N    "AutoProcessData".GripperCode_R2[3]:="KeyenceSR1000Ctrl_806A1DB".sHMI.Status.CurrentCode
   END_STEP
   TRANSITION Trans331 FROM DataMove_16 TO RobotScanGripPos3Comp_1   // T378
      := "AlwaysTRUE";
   END_TRANSITION
   STEP RobotScanGripPos3Comp_1:   // S378, max time T#10S, warning time T#7S
              R    "KukaRobot2_CtrlDB".sPLCtoROB.User.Cycle.DI307_ScanPartFinish
              N    "KukaRobot2_CtrlDB".sPLCtoROB.User.Cycle.DI306_ScanPartComplete
   END_STEP
   TRANSITION Trans332 FROM RobotScanGripPos3Comp_1 TO WaitRobotScanGripPos4Reach_1   // T379
      := NOT "KukaRobot2_CtrlDB".sROBtoPLC.User.Cycle.DO309_ScanPos3Reach;
   END_TRANSITION
   STEP WaitRobotScanGripPos4Reach_1:   // S383, max time T#10S, warning time T#7S
   END_STEP
   TRANSITION Trans333 FROM WaitRobotScanGripPos4Reach_1 TO "Check reader Ready_17"   // T381
      := "KukaRobot2_CtrlDB".sROBtoPLC.User.Cycle.DO310_ScanPos4Reach;
   END_TRANSITION
   STEP "Check reader Ready_17":   // S385, max time T#10S, warning time T#7S
   END_STEP
   TRANSITION Trans676 FROM "Check reader Ready_17" TO "Start 11st reading_5"   // T635
      := "KeyenceSR1000Ctrl_806A1DB".oReady;
   END_TRANSITION
   STEP "Start 11st reading_5":   // S386, max time T#10S, warning time T#7S
          S1  S    "KeyenceSR1000Ctrl_806A1DB".ioAutoTrigger
   END_STEP
   TRANSITION Trans677 FROM "Start 11st reading_5" TO "Wait reading complete_17"   // T638
      := NOT "KeyenceSR1000Ctrl_806A1DB".sHMI.Status.Ready;
   END_TRANSITION
   STEP "Wait reading complete_17":   // S388, max time T#10S, warning time T#7S
   END_STEP
   TRANSITION ReadOK_17 FROM "Wait reading complete_17" TO DataMove_17   // T382
      := "KeyenceSR1000Ctrl_806A1DB".sHMI.Status.Complete;
   END_TRANSITION
   STEP DataMove_17:   // S389, max time T#10S, warning time T#7S
              N    "AutoProcessData".GripperCode_R2[4]:="KeyenceSR1000Ctrl_806A1DB".sHMI.Status.CurrentCode
   END_STEP
   TRANSITION Trans334 FROM DataMove_17 TO RobotScanGripPos4Comp_1   // T384
      := "AlwaysTRUE";
   END_TRANSITION
   STEP RobotScanGripPos4Comp_1:   // S391, max time T#10S, warning time T#7S
              N    "KukaRobot2_CtrlDB".sPLCtoROB.User.Cycle.DI307_ScanPartFinish
              N    "KukaRobot2_CtrlDB".sPLCtoROB.User.Cycle.DI306_ScanPartComplete
   END_STEP
   TRANSITION Trans335 FROM RobotScanGripPos4Comp_1 TO Robot2CheckScanResult   // T385
      := "KukaRobot2_CtrlDB".sROBtoPLC.User.Cycle.DO306_GripScanFinish;
   END_TRANSITION
   STEP StartRobotScanGripperCode:   // S363, max time T#10S, warning time T#7S
              N    "AutoProcessControl".Robot_2.GripScanRequest
   END_STEP
   TRANSITION Trans684 FROM StartRobotScanGripperCode TO RobotScanGripperReachPos1   // T616
      := "KukaRobot2_CtrlDB".sROBtoPLC.User.Cycle.DO305_GripScanInside AND NOT "KukaRobot2_CtrlDB".sROBtoPLC.User.Cycle.DO306_GripScanFinish;
   END_TRANSITION
   STEP RobotScanGripperReachPos1:   // S364, max time T#10S, warning time T#7S
   END_STEP
   TRANSITION Trans685 FROM RobotScanGripperReachPos1 TO "Check reader Ready_14"   // T673
      := "KukaRobot2_CtrlDB".sROBtoPLC.User.Cycle.DO307_ScanPos1Reach;
   END_TRANSITION
   STEP Robot2CheckScanStatus:   // S410, max time T#10S, warning time T#7S
   END_STEP
   TRANSITION "317GripScanng" FROM Robot2CheckScanStatus TO StartRobotScanGripperCode   // T317
      := NOT "AutoProcessData".GlobalData.Robot2GripperCodeOKFlag;
   END_TRANSITION
   TRANSITION "319GripScanOK" FROM Robot2CheckScanStatus TO Robot2CheckScanResult   // T319
      := "AutoProcessData".GlobalData.Robot2GripperCodeOKFlag;
   END_TRANSITION

